  MoveC 574 to (267.87, -55.04, -8.35) mm, rotated rx 180 ry 0 rz 0 deg; joints [19.535, -64.731, 149.655, 19.627, -84.348, -1.431] to (268.06, -55.49, -8.35) mm, rotated rx 180 ry 0 rz 0 deg; joints [19.512, -64.74, 149.678, 19.605, -84.361, -1.424]
  MoveL 575 to (268.06, -80.89, -8.35) mm, rotated rx 180 ry 0 rz 0 deg; joints [18.023, -64.948, 150.269, 18.098, -84.683, -1.18]
  MoveL 576 to (217.26, -80.89, -8.35) mm, rotated rx -180 ry 0 rz 0 deg; joints [17.095, -63.534, 146.744, 17.235, -82.641, -1.736]
  MoveL 577 to (217.26, -30.09, -8.35) mm, rotated rx -180 ry 0 rz 0 deg; joints [19.918, -63.093, 145.562, 20.113, -82.053, -2.311]
  MoveL 578 to (268.06, -30.09, -8.35) mm, rotated rx 180 ry 0 rz 0 deg; joints [20.974, -64.512, 149.041, 21.088, -84.024, -1.694]
  MoveL 579 to (268.06, -55.49, -8.35) mm, rotated rx 180 ry 0 rz 0 deg; joints [19.512, -64.74, 149.678, 19.605, -84.361, -1.424]
  MoveC 580 to (267.87, -55.94, -8.35) mm, rotated rx -180 ry 0 rz 0 deg; joints [19.482, -64.739, 149.677, 19.575, -84.359, -1.422] to (267.42, -56.12, -8.35) mm, rotated rx -180 ry 0 rz 0 deg; joints [19.462, -64.728, 149.65, 19.555, -84.344, -1.425]
  MoveL 581 to (266.79, -56.12, -8.35) mm, rotated rx 180 ry 0 rz 0 deg; joints [19.449, -64.711, 149.607, 19.543, -84.319, -1.433]
  MoveC 582 to (266.34, -56.12, -8.16) mm, rotated rx 180 ry 0 rz 0 deg; joints [19.44, -64.717, 149.577, 19.535, -84.284, -1.445] to (266.15, -56.12, -7.72) mm, rotated rx -180 ry 0 rz 0 deg; joints [19.436, -64.757, 149.566, 19.532, -84.236, -1.461]
  Set speed (500.0 mm/s)
  MoveL 583 to (266.15, -56.12, 6) mm, rotated rx 180 ry 0 rz 0 deg; joints [19.428, -66.123, 149.601, 19.574, -82.982, -1.909]
  MoveL 584 to (139.15, -54.85, 6) mm, rotated rx -180 ry 0 rz 0 deg; joints [17.193, -62.179, 140.681, 17.573, -78.154, -3.178]
  Set speed (25.4 mm/s)
  MoveL 585 to (139.15, -54.85, -3.54) mm, rotated rx 180 ry 0 rz 0 deg; joints [17.198, -61.393, 140.662, 17.531, -78.886, -2.943]
  MoveC 586 to (139.34, -54.85, -3.99) mm, rotated rx 180 ry 0 rz 0 deg; joints [17.201, -61.361, 140.675, 17.531, -78.928, -2.93] to (139.79, -54.85, -4.17) mm, rotated rx 180 ry 0 rz 0 deg; joints [17.208, -61.36, 140.706, 17.537, -78.96, -2.921]
  Set speed (50.8 mm/s)
  MoveL 587 to (140.42, -54.85, -4.17) mm, rotated rx -180 ry 0 rz 0 deg; joints [17.219, -61.38, 140.752, 17.546, -78.985, -2.915]
  MoveC 588 to (140.87, -55.04, -4.17) mm, rotated rx -180 ry 0 rz 0 deg; joints [17.216, -61.395, 140.788, 17.542, -79.004, -2.909] to (141.06, -55.49, -4.17) mm, rotated rx -180 ry 0 rz 0 deg; joints [17.196, -61.405, 140.811, 17.521, -79.016, -2.901]
  MoveL 589 to (141.06, -80.89, -4.17) mm, rotated rx 180 ry 0 rz 0 deg; joints [15.863, -61.621, 141.351, 16.147, -79.257, -2.57]
  MoveL 590 to (90.26, -80.89, -4.17) mm, rotated rx 180 ry 0 rz 0 deg; joints [15.134, -60.003, 137.665, 15.522, -77.228, -3.006]
  MoveL 591 to (90.26, -30.09, -4.17) mm, rotated rx 180 ry 0 rz 0 deg; joints [17.675, -59.554, 136.575, 18.167, -76.776, -3.743]
  MoveL 592 to (141.06, -30.09, -4.18) mm, rotated rx -180 ry 0 rz 0 deg; joints [18.51, -61.17, 140.228, 18.879, -78.762, -3.249]
  MoveL 593 to (141.06, -55.49, -4.17) mm, rotated rx -180 ry 0 rz 0 deg; joints [17.196, -61.405, 140.811, 17.521, -79.016, -2.901]
  MoveC 594 to (140.87, -55.94, -4.17) mm, rotated rx 180 ry 0 rz 0 deg; joints [17.169, -61.403, 140.808, 17.494, -79.013, -2.897] to (140.42, -56.12, -4.18) mm, rotated rx 180 ry 0 rz 0 deg; joints [17.152, -61.391, 140.78, 17.478, -78.997, -2.898]
  MoveL 595 to (139.79, -56.12, -4.18) mm, rotated rx 180 ry 0 rz 0 deg; joints [17.142, -61.371, 140.734, 17.469, -78.972, -2.904]
  MoveC 596 to (139.34, -56.12, -3.99) mm, rotated rx -180 ry 0 rz 0 deg; joints [17.135, -61.373, 140.703, 17.463, -78.94, -2.913] to (139.15, -56.12, -3.54) mm, rotated rx -180 ry 0 rz 0 deg; joints [17.132, -61.404, 140.69, 17.463, -78.899, -2.926]
  Set speed (500.0 mm/s)
  MoveL 597 to (139.15, -56.12, 5) mm, rotated rx -180 ry 0 rz 0 deg; joints [17.128, -62.108, 140.708, 17.5, -78.243, -3.136]
  MoveL 598 to (139.15, -54.85, 5) mm, rotated rx -180 ry 0 rz 0 deg; joints [17.194, -62.097, 140.68, 17.568, -78.231, -3.153]
  Set speed (25.4 mm/s)
  MoveL 599 to (139.15, -54.85, 1.82) mm, rotated rx -180 ry 0 rz 0 deg; joints [17.195, -61.835, 140.674, 17.554, -78.475, -3.075]
  MoveL 600 to (139.15, -54.85, -7.71) mm, rotated rx -180 ry 0 rz 0 deg; joints [17.2, -61.047, 140.651, 17.513, -79.205, -2.841]
  MoveC 601 to (139.34, -54.85, -8.16) mm, rotated rx -180 ry 0 rz 0 deg; joints [17.203, -61.016, 140.663, 17.514, -79.247, -2.828] to (139.79, -54.85, -8.35) mm, rotated rx -180 ry 0 rz 0 deg; joints [17.21, -61.014, 140.695, 17.52, -79.279, -2.819]
  Set speed (50.8 mm/s)
  MoveL 602 to (140.42, -54.85, -8.35) mm, rotated rx -180 ry 0 rz 0 deg; joints [17.221, -61.034, 140.74, 17.529, -79.304, -2.813]
  MoveC 603 to (140.87, -55.04, -8.35) mm, rotated rx 180 ry 0 rz 0 deg; joints [17.218, -61.049, 140.776, 17.525, -79.324, -2.806] to (141.06, -55.49, -8.35) mm, rotated rx 180 ry 0 rz 0 deg; joints [17.198, -61.059, 140.8, 17.503, -79.336, -2.799]
  MoveL 604 to (141.06, -80.89, -8.35) mm, rotated rx -180 ry 0 rz 0 deg; joints [15.865, -61.271, 141.339, 16.132, -79.582, -2.475]
  MoveL 605 to (90.26, -80.89, -8.35) mm, rotated rx -180 ry 0 rz 0 deg; joints [15.136, -59.676, 137.654, 15.505, -77.533, -2.92]
  MoveL 606 to (90.26, -30.09, -8.35) mm, rotated rx -180 ry 0 rz 0 deg; joints [17.677, -59.233, 136.564, 18.146, -77.071, -3.645]
  MoveL 607 to (141.06, -30.09, -8.35) mm, rotated rx 180 ry 0 rz 0 deg; joints [18.512, -60.828, 140.217, 18.86, -79.076, -3.141]
  MoveL 608 to (141.06, -55.49, -8.35) mm, rotated rx 180 ry 0 rz 0 deg; joints [17.198, -61.059, 140.8, 17.503, -79.336, -2.799]
  MoveC 609 to (140.87, -55.94, -8.35) mm, rotated rx -180 ry 0 rz 0 deg; joints [17.171, -61.057, 140.796, 17.477, -79.333, -2.795] to (140.42, -56.12, -8.35) mm, rotated rx 180 ry 0 rz 0 deg; joints [17.155, -61.045, 140.768, 17.46, -79.317, -2.796]
  MoveL 610 to (139.79, -56.12, -8.35) mm, rotated rx 180 ry 0 rz 0 deg; joints [17.144, -61.025, 140.723, 17.452, -79.291, -2.803]
  MoveC 611 to (139.34, -56.12, -8.16) mm, rotated rx -180 ry 0 rz 0 deg; joints [17.137, -61.027, 140.691, 17.446, -79.259, -2.811] to (139.15, -56.12, -7.72) mm, rotated rx -180 ry 0 rz 0 deg; joints [17.134, -61.058, 140.679, 17.445, -79.218, -2.824]
  Set speed (500.0 mm/s)
  MoveL 612 to (139.15, -56.12, 6) mm, rotated rx -180 ry 0 rz 0 deg; joints [17.127, -62.191, 140.709, 17.505, -78.166, -3.16]
  MoveL 613 to (139.15, -235.88, 6) mm, rotated rx -180 ry 0 rz 0 deg; joints [7.369, -63.345, 143.558, 7.492, -79.426, -0.998]
  Set speed (25.4 mm/s)
  MoveL 614 to (139.15, -235.88, -3.54) mm, rotated rx 180 ry 0 rz 0 deg; joints [7.373, -62.513, 143.538, 7.477, -80.231, -0.891]
  MoveC 615 to (139.34, -235.88, -3.99) mm, rotated rx -180 ry 0 rz 0 deg; joints [7.374, -62.48, 143.551, 7.477, -80.276, -0.885] to (139.79, -235.88, -4.17) mm, rotated rx -180 ry 0 rz 0 deg; joints [7.378, -62.477, 143.583, 7.48, -80.311, -0.881]
  Set speed (50.8 mm/s)
  MoveL 616 to (140.42, -235.88, -4.18) mm, rotated rx -180 ry 0 rz 0 deg; joints [7.382, -62.497, 143.63, 7.484, -80.337, -0.878]
  MoveC 617 to (140.87, -236.07, -4.18) mm, rotated rx -180 ry 0 rz 0 deg; joints [7.375, -62.512, 143.665, 7.476, -80.357, -0.874] to (141.06, -236.52, -4.18) mm, rotated rx -180 ry 0 rz 0 deg; joints [7.351, -62.519, 143.683, 7.452, -80.367, -0.869]
  MoveL 618 to (141.06, -261.92, -4.17) mm, rotated rx 180 ry 0 rz 0 deg; joints [5.92, -62.597, 143.899, 5.998, -80.48, -0.633]
  MoveL 619 to (90.26, -261.92, -4.18) mm, rotated rx -180 ry 0 rz 0 deg; joints [5.637, -60.978, 140.132, 5.751, -78.337, -0.808]
  MoveL 620 to (90.26, -211.12, -4.17) mm, rotated rx 180 ry 0 rz 0 deg; joints [8.357, -60.803, 139.668, 8.536, -78.115, -1.37]
  MoveL 621 to (141.06, -211.12, -4.17) mm, rotated rx -180 ry 0 rz 0 deg; joints [8.773, -62.422, 143.419, 8.898, -80.234, -1.115]
  MoveL 622 to (141.06, -236.52, -4.18) mm, rotated rx -180 ry 0 rz 0 deg; joints [7.351, -62.519, 143.683, 7.452, -80.367, -0.869]
  MoveC 623 to (140.87, -236.97, -4.17) mm, rotated rx -180 ry 0 rz 0 deg; joints [7.325, -62.515, 143.673, 7.425, -80.362, -0.866] to (140.42, -237.16, -4.17) mm, rotated rx -180 ry 0 rz 0 deg; joints [7.311, -62.502, 143.642, 7.412, -80.344, -0.866]
  MoveL 624 to (139.79, -237.16, -4.17) mm, rotated rx 180 ry 0 rz 0 deg; joints [7.306, -62.482, 143.595, 7.408, -80.317, -0.869]
  MoveC 625 to (139.34, -237.15, -3.99) mm, rotated rx -180 ry 0 rz 0 deg; joints [7.303, -62.484, 143.563, 7.405, -80.282, -0.873] to (139.15, -237.15, -3.54) mm, rotated rx -180 ry 0 rz 0 deg; joints [7.302, -62.517, 143.55, 7.404, -80.237, -0.879]
  Set speed (500.0 mm/s)
  MoveL 626 to (139.15, -237.16, 5) mm, rotated rx 180 ry 0 rz 0 deg; joints [7.298, -63.263, 143.569, 7.418, -79.516, -0.973]
  MoveL 627 to (139.15, -235.88, 5) mm, rotated rx -180 ry 0 rz 0 deg; joints [7.37, -63.258, 143.557, 7.491, -79.51, -0.987]
  Set speed (25.4 mm/s)
  MoveL 628 to (139.15, -235.89, 1.82) mm, rotated rx 180 ry 0 rz 0 deg; joints [7.371, -62.981, 143.551, 7.485, -79.779, -0.951]
  MoveL 629 to (139.15, -235.88, -7.71) mm, rotated rx -180 ry 0 rz 0 deg; joints [7.374, -62.148, 143.526, 7.471, -80.581, -0.845]
  MoveC 630 to (139.34, -235.88, -8.16) mm, rotated rx -180 ry 0 rz 0 deg; joints [7.376, -62.114, 143.539, 7.471, -80.627, -0.839] to (139.79, -235.89, -8.35) mm, rotated rx 180 ry 0 rz 0 deg; joints [7.379, -62.111, 143.571, 7.474, -80.661, -0.835]
  Set speed (50.8 mm/s)
  MoveL 631 to (140.42, -235.88, -8.35) mm, rotated rx -180 ry 0 rz 0 deg; joints [7.384, -62.131, 143.618, 7.478, -80.688, -0.832]
  MoveC 632 to (140.87, -236.07, -8.35) mm, rotated rx -180 ry 0 rz 0 deg; joints [7.377, -62.145, 143.652, 7.47, -80.708, -0.828] to (141.06, -236.52, -8.35) mm, rotated rx -180 ry 0 rz 0 deg; joints [7.353, -62.153, 143.67, 7.446, -80.718, -0.823]
  MoveL 633 to (141.06, -261.92, -8.35) mm, rotated rx -180 ry 0 rz 0 deg; joints [5.921, -62.229, 143.887, 5.993, -80.834, -0.596]
  MoveL 634 to (90.26, -261.92, -8.35) mm, rotated rx -180 ry 0 rz 0 deg; joints [5.638, -60.636, 140.12, 5.746, -78.666, -0.775]
  MoveL 635 to (90.26, -211.12, -8.35) mm, rotated rx 180 ry 0 rz 0 deg; joints [8.358, -60.464, 139.657, 8.528, -78.439, -1.321]
  MoveL 636 to (141.06, -211.12, -8.35) mm, rotated rx 180 ry 0 rz 0 deg; joints [8.775, -62.058, 143.407, 8.891, -80.582, -1.06]
  MoveL 637 to (141.06, -236.52, -8.35) mm, rotated rx -180 ry 0 rz 0 deg; joints [7.353, -62.153, 143.67, 7.446, -80.718, -0.823]
  MoveC 638 to (140.87, -236.97, -8.35) mm, rotated rx 180 ry 0 rz 0 deg; joints [7.326, -62.148, 143.661, 7.419, -80.713, -0.82] to (140.42, -237.16, -8.35) mm, rotated rx -180 ry 0 rz 0 deg; joints [7.313, -62.135, 143.63, 7.406, -80.695, -0.82]
  MoveL 639 to (139.79, -237.15, -8.35) mm, rotated rx -180 ry 0 rz 0 deg; joints [7.308, -62.116, 143.583, 7.402, -80.668, -0.823]
  MoveC 640 to (139.34, -237.15, -8.16) mm, rotated rx 180 ry 0 rz 0 deg; joints [7.305, -62.118, 143.551, 7.399, -80.633, -0.827] to (139.15, -237.16, -7.72) mm, rotated rx -180 ry 0 rz 0 deg; joints [7.303, -62.152, 143.538, 7.398, -80.587, -0.833]
  Set speed (500.0 mm/s)
  MoveL 641 to (139.15, -237.16, 6) mm, rotated rx -180 ry 0 rz 0 deg; joints [7.298, -63.35, 143.57, 7.42, -79.431, -0.985]
  MoveL 642 to (266.15, -235.88, 6) mm, rotated rx -180 ry 0 rz 0 deg; joints [8.42, -67.287, 152.736, 8.452, -84.629, -0.396]
  Set speed (25.4 mm/s)
  MoveL 643 to (266.15, -235.89, -3.54) mm, rotated rx 180 ry 0 rz 0 deg; joints [8.424, -66.261, 152.712, 8.444, -85.619, -0.249]
  MoveC 644 to (266.34, -235.88, -3.99) mm, rotated rx -180 ry 0 rz 0 deg; joints [8.426, -66.218, 152.723, 8.445, -85.674, -0.241] to (266.79, -235.89, -4.17) mm, rotated rx -180 ry 0 rz 0 deg; joints [8.43, -66.21, 152.755, 8.449, -85.712, -0.235]
  Set speed (50.8 mm/s)
  MoveL 645 to (267.42, -235.89, -4.17) mm, rotated rx -180 ry 0 rz 0 deg; joints [8.436, -66.228, 152.8, 8.455, -85.74, -0.231]
  MoveC 646 to (267.87, -236.07, -4.18) mm, rotated rx -180 ry 0 rz 0 deg; joints [8.429, -66.241, 152.834, 8.447, -85.76, -0.228] to (268.06, -236.52, -4.17) mm, rotated rx 180 ry 0 rz 0 deg; joints [8.402, -66.247, 152.852, 8.42, -85.772, -0.225]
  MoveL 647 to (268.06, -261.92, -4.18) mm, rotated rx -180 ry 0 rz 0 deg; joints [6.77, -66.321, 153.092, 6.782, -85.924, -0.109]
  MoveL 648 to (217.26, -261.92, -4.18) mm, rotated rx 180 ry 0 rz 0 deg; joints [6.402, -64.892, 149.45, 6.436, -83.722, -0.337]
  MoveL 649 to (217.26, -211.12, -4.18) mm, rotated rx -180 ry 0 rz 0 deg; joints [9.482, -64.721, 148.941, 9.54, -83.43, -0.684]
  MoveL 650 to (268.06, -211.12, -4.17) mm, rotated rx 180 ry 0 rz 0 deg; joints [10.02, -66.154, 152.56, 10.045, -85.591, -0.354]
  MoveL 651 to (268.06, -236.52, -4.17) mm, rotated rx 180 ry 0 rz 0 deg; joints [8.402, -66.247, 152.852, 8.42, -85.772, -0.225]
  MoveC 652 to (267.87, -236.97, -4.17) mm, rotated rx -180 ry 0 rz 0 deg; joints [8.371, -66.244, 152.843, 8.389, -85.766, -0.224] to (267.42, -237.15, -4.18) mm, rotated rx -180 ry 0 rz 0 deg; joints [8.355, -66.232, 152.813, 8.373, -85.748, -0.225]
  MoveL 653 to (266.79, -237.15, -4.18) mm, rotated rx -180 ry 0 rz 0 deg; joints [8.349, -66.215, 152.768, 8.368, -85.721, -0.229]
  MoveC 654 to (266.34, -237.15, -3.99) mm, rotated rx 180 ry 0 rz 0 deg; joints [8.345, -66.222, 152.737, 8.364, -85.682, -0.234] to (266.15, -237.16, -3.54) mm, rotated rx 180 ry 0 rz 0 deg; joints [8.343, -66.266, 152.725, 8.362, -85.627, -0.242]
  Set speed (500.0 mm/s)
  MoveL 655 to (266.15, -237.16, 5) mm, rotated rx -180 ry 0 rz 0 deg; joints [8.339, -67.184, 152.747, 8.37, -84.741, -0.373]
  MoveL 656 to (266.15, -235.89, 5) mm, rotated rx -180 ry 0 rz 0 deg; joints [8.42, -67.18, 152.734, 8.451, -84.733, -0.38]
  Set speed (25.4 mm/s)
  MoveL 657 to (266.15, -235.88, 1.82) mm, rotated rx -180 ry 0 rz 0 deg; joints [8.422, -66.839, 152.727, 8.448, -85.063, -0.331]
  MoveL 658 to (266.15, -235.89, -7.71) mm, rotated rx 180 ry 0 rz 0 deg; joints [8.426, -65.811, 152.697, 8.441, -86.05, -0.185]
  MoveC 659 to (266.34, -235.89, -8.16) mm, rotated rx -180 ry 0 rz 0 deg; joints [8.428, -65.768, 152.709, 8.442, -86.104, -0.177] to (266.79, -235.88, -8.35) mm, rotated rx -180 ry 0 rz 0 deg; joints [8.432, -65.76, 152.74, 8.446, -86.143, -0.171]
  Set speed (50.8 mm/s)
  MoveL 660 to (267.42, -235.88, -8.35) mm, rotated rx -180 ry 0 rz 0 deg; joints [8.438, -65.777, 152.785, 8.452, -86.171, -0.167]
  MoveC 661 to (267.87, -236.07, -8.35) mm, rotated rx 180 ry 0 rz 0 deg; joints [8.431, -65.789, 152.819, 8.444, -86.193, -0.164] to (268.06, -236.52, -8.35) mm, rotated rx 180 ry 0 rz 0 deg; joints [8.404, -65.795, 152.837, 8.417, -86.204, -0.161]
  MoveL 662 to (268.06, -261.92, -8.35) mm, rotated rx -180 ry 0 rz 0 deg; joints [6.772, -65.866, 153.077, 6.781, -86.361, -0.057]
  MoveL 663 to (217.26, -261.92, -8.35) mm, rotated rx 180 ry 0 rz 0 deg; joints [6.404, -64.477, 149.436, 6.433, -84.122, -0.292]
  MoveL 664 to (217.26, -211.12, -8.35) mm, rotated rx 180 ry 0 rz 0 deg; joints [9.483, -64.31, 148.928, 9.534, -83.822, -0.618]
  MoveL 665 to (268.06, -211.12, -8.35) mm, rotated rx -180 ry 0 rz 0 deg; joints [10.022, -65.706, 152.546, 10.041, -86.018, -0.278]
  MoveL 666 to (268.06, -236.52, -8.35) mm, rotated rx -180 ry 0 rz 0 deg; joints [8.404, -65.795, 152.837, 8.417, -86.204, -0.161]
  MoveC 667 to (267.87, -236.97, -8.35) mm, rotated rx -180 ry 0 rz 0 deg; joints [8.373, -65.792, 152.828, 8.387, -86.199, -0.16] to (267.42, -237.15, -8.35) mm, rotated rx -180 ry 0 rz 0 deg; joints [8.357, -65.781, 152.798, 8.371, -86.18, -0.162]
  MoveL 668 to (266.79, -237.15, -8.35) mm, rotated rx -180 ry 0 rz 0 deg; joints [8.351, -65.764, 152.753, 8.365, -86.152, -0.165]
  MoveC 669 to (266.34, -237.15, -8.16) mm, rotated rx -180 ry 0 rz 0 deg; joints [8.347, -65.772, 152.722, 8.361, -86.113, -0.171] to (266.15, -237.15, -7.72) mm, rotated rx 180 ry 0 rz 0 deg; joints [8.345, -65.815, 152.711, 8.36, -86.059, -0.179]
  Set speed (500.0 mm/s)
  MoveL 670 to (266.15, -237.15, 6) mm, rotated rx -180 ry 0 rz 0 deg; joints [8.339, -67.291, 152.749, 8.371, -84.636, -0.388]
  MoveL 671 to (393.15, -235.89, 6) mm, rotated rx 180 ry 0 rz 30 deg; joints [20.408, -68.62, 155.616, 50.482, -87.198, -2.516]
  Set speed (25.4 mm/s)
  MoveL 672 to (393.15, -235.88, -3.54) mm, rotated rx -180 ry 0 rz 30 deg; joints [20.414, -67.513, 155.591, 50.452, -87.887, -1.681]
  MoveC 673 to (393.34, -235.89, -3.99) mm, rotated rx 180 ry 0 rz 30 deg; joints [20.419, -67.465, 155.602, 50.455, -87.924, -1.636] to (393.79, -235.88, -4.17) mm, rotated rx -180 ry 0 rz 30 deg; joints [20.43, -67.455, 155.631, 50.465, -87.95, -1.605]
  Set speed (50.8 mm/s)
  MoveL 674 to (394.42, -235.88, -4.18) mm, rotated rx -180 ry 0 rz 30 deg; joints [20.445, -67.47, 155.674, 50.479, -87.967, -1.585]
  MoveC 675 to (394.87, -236.07, -4.17) mm, rotated rx -180 ry 0 rz 30 deg; joints [20.443, -67.483, 155.708, 50.478, -87.981, -1.568] to (395.06, -236.52, -4.18) mm, rotated rx -180 ry 0 rz 30 deg; joints [20.419, -67.491, 155.732, 50.453, -87.99, -1.555]
  MoveL 676 to (395.06, -261.92, -4.17) mm, rotated rx -180 ry 0 rz 30 deg; joints [18.79, -67.683, 156.338, 48.813, -88.225, -1.211]
  MoveL 677 to (344.26, -261.92, -4.18) mm, rotated rx -180 ry 0 rz 30 deg; joints [17.731, -66.386, 152.89, 47.824, -86.761, -2.789]
  MoveL 678 to (344.26, -211.12, -4.17) mm, rotated rx 180 ry 0 rz 0 deg; joints [10.952, -68.118, 157.906, 10.948, -88.922, 0.232]
  MoveL 679 to (395.06, -211.12, -4.18) mm, rotated rx -180 ry 0 rz 30 deg; joints [22.015, -67.278, 155.078, 52.062, -87.757, -1.935]
  MoveL 680 to (395.06, -236.52, -4.17) mm, rotated rx -180 ry 0 rz 30 deg; joints [20.419, -67.491, 155.732, 50.453, -87.99, -1.555]
  MoveC 681 to (394.87, -236.97, -4.18) mm, rotated rx 180 ry 0 rz 30 deg; joints [20.386, -67.49, 155.731, 50.42, -87.989, -1.555] to (394.42, -237.15, -4.18) mm, rotated rx -180 ry 0 rz 30 deg; joints [20.364, -67.48, 155.705, 50.398, -87.979, -1.567]
  MoveL 682 to (393.79, -237.16, -4.18) mm, rotated rx 180 ry 0 rz 30 deg; joints [20.349, -67.465, 155.663, 50.384, -87.961, -1.587]
  MoveC 683 to (393.34, -237.15, -3.99) mm, rotated rx -180 ry 0 rz 30 deg; joints [20.338, -67.475, 155.634, 50.374, -87.936, -1.618] to (393.15, -237.15, -3.54) mm, rotated rx 180 ry 0 rz 30 deg; joints [20.334, -67.523, 155.623, 50.371, -87.898, -1.663]
  Set speed (500.0 mm/s)
  MoveL 684 to (393.15, -237.16, 5) mm, rotated rx -180 ry 0 rz 30 deg; joints [20.328, -68.515, 155.646, 50.397, -87.28, -2.41]
  MoveL 685 to (393.15, -235.88, 5) mm, rotated rx 180 ry 0 rz 30 deg; joints [20.408, -68.504, 155.614, 50.478, -87.27, -2.428]
  Set speed (25.4 mm/s)
  MoveL 686 to (393.15, -235.88, 1.82) mm, rotated rx -180 ry 0 rz 30 deg; joints [20.411, -68.136, 155.607, 50.468, -87.5, -2.15]
  MoveL 687 to (393.15, -235.89, -7.71) mm, rotated rx -180 ry 0 rz 30 deg; joints [20.417, -67.027, 155.576, 50.443, -88.187, -1.318]
  MoveC 688 to (393.34, -235.89, -8.16) mm, rotated rx 180 ry 0 rz 30 deg; joints [20.422, -66.979, 155.587, 50.446, -88.224, -1.272] to (393.79, -235.88, -8.35) mm, rotated rx -180 ry 0 rz 30 deg; joints [20.432, -66.968, 155.616, 50.456, -88.25, -1.242]
  Set speed (50.8 mm/s)
  MoveL 689 to (394.42, -235.89, -8.35) mm, rotated rx 180 ry 0 rz 30 deg; joints [20.447, -66.983, 155.658, 50.47, -88.267, -1.221]
  MoveC 690 to (394.87, -236.07, -8.35) mm, rotated rx -180 ry 0 rz 30 deg; joints [20.446, -66.995, 155.693, 50.468, -88.282, -1.203] to (395.06, -236.52, -8.35) mm, rotated rx -180 ry 0 rz 30 deg; joints [20.422, -67.003, 155.717, 50.444, -88.291, -1.191]
  MoveL 691 to (395.06, -261.92, -8.35) mm, rotated rx -180 ry 0 rz 30 deg; joints [18.792, -67.187, 156.322, 48.805, -88.541, -0.85]
  MoveL 692 to (344.26, -261.92, -8.35) mm, rotated rx -180 ry 0 rz 30 deg; joints [17.733, -65.934, 152.875, 47.809, -87.055, -2.465]
  MoveL 693 to (344.26, -211.12, -8.35) mm, rotated rx -180 ry 0 rz 0 deg; joints [10.954, -67.598, 157.889, 10.949, -89.416, 0.328]
  MoveL 694 to (395.06, -211.12, -8.35) mm, rotated rx -180 ry 0 rz 30 deg; joints [22.018, -66.799, 155.062, 52.051, -88.042, -1.568]
  MoveL 695 to (395.06, -236.52, -8.35) mm, rotated rx -180 ry 0 rz 30 deg; joints [20.422, -67.003, 155.717, 50.444, -88.291, -1.191]
  MoveC 696 to (394.87, -236.97, -8.35) mm, rotated rx -180 ry 0 rz 30 deg; joints [20.389, -67.002, 155.715, 50.411, -88.291, -1.191] to (394.42, -237.15, -8.35) mm, rotated rx 180 ry 0 rz 30 deg; joints [20.367, -66.993, 155.69, 50.389, -88.28, -1.203]
  MoveL 697 to (393.79, -237.15, -8.35) mm, rotated rx -180 ry 0 rz 30 deg; joints [20.352, -66.978, 155.648, 50.375, -88.262, -1.224]
  MoveC 698 to (393.34, -237.15, -8.16) mm, rotated rx -180 ry 0 rz 30 deg; joints [20.341, -66.989, 155.618, 50.365, -88.236, -1.254] to (393.15, -237.15, -7.72) mm, rotated rx 180 ry 0 rz 30 deg; joints [20.336, -67.037, 155.608, 50.362, -88.199, -1.3]
  Set speed (500.0 mm/s)
  MoveL 699 to (393.15, -237.16, 6) mm, rotated rx -180 ry 0 rz 30 deg; joints [20.327, -68.631, 155.648, 50.401, -87.207, -2.498]
  MoveL 700 to (393.15, -422.22, 6) mm, rotated rx -180 ry 0 rz 60 deg; joints [14.177, -65.672, 148.72, 74.367, -87.443, -7.311]
  Set speed (25.4 mm/s)
  MoveL 701 to (393.15, -422.22, -3.54) mm, rotated rx -180 ry 0 rz 60 deg; joints [14.182, -64.742, 148.698, 74.335, -87.688, -6.436]
  MoveC 702 to (393.34, -422.22, -3.99) mm, rotated rx -180 ry 0 rz 60 deg; joints [14.185, -64.704, 148.71, 74.336, -87.702, -6.387] to (393.79, -422.22, -4.17) mm, rotated rx -180 ry 0 rz 60 deg; joints [14.192, -64.698, 148.741, 74.342, -87.713, -6.353]
  Set speed (50.8 mm/s)
  MoveL 703 to (394.42, -422.22, -4.18) mm, rotated rx -180 ry 0 rz 60 deg; joints [14.201, -64.717, 148.786, 74.35, -87.721, -6.327]
  MoveC 704 to (394.87, -422.41, -4.18) mm, rotated rx -180 ry 0 rz 60 deg; joints [14.197, -64.731, 148.821, 74.345, -87.726, -6.307] to (395.06, -422.86, -4.17) mm, rotated rx -180 ry 0 rz 60 deg; joints [14.173, -64.739, 148.842, 74.321, -87.727, -6.294]
  MoveL 705 to (395.06, -448.26, -4.17) mm, rotated rx -180 ry 0 rz 60 deg; joints [12.665, -64.892, 149.27, 72.807, -87.66, -5.987]
  MoveL 706 to (344.26, -448.26, -4.17) mm, rotated rx -180 ry 0 rz 30 deg; joints [5.639, -67.24, 155.598, 35.664, -87.777, -1.156]
  MoveL 707 to (344.26, -397.46, -4.18) mm, rotated rx 180 ry 0 rz 30 deg; joints [9.034, -67.111, 155.137, 39.069, -87.578, -1.443]
  MoveL 708 to (395.06, -397.46, -4.17) mm, rotated rx 180 ry 0 rz 60 deg; joints [15.662, -64.566, 148.367, 75.814, -87.801, -6.627]
  MoveL 709 to (395.06, -422.86, -4.17) mm, rotated rx -180 ry 0 rz 60 deg; joints [14.173, -64.739, 148.842, 74.321, -87.727, -6.294]
  MoveC 710 to (394.87, -423.31, -4.18) mm, rotated rx -180 ry 0 rz 60 deg; joints [14.144, -64.737, 148.837, 74.292, -87.724, -6.296] to (394.42, -423.49, -4.18) mm, rotated rx 180 ry 0 rz 60 deg; joints [14.126, -64.725, 148.809, 74.275, -87.717, -6.311]
  MoveL 711 to (393.79, -423.49, -4.17) mm, rotated rx -180 ry 0 rz 60 deg; joints [14.117, -64.707, 148.764, 74.266, -87.709, -6.337]
  MoveC 712 to (393.34, -423.49, -3.99) mm, rotated rx -180 ry 0 rz 60 deg; joints [14.11, -64.712, 148.733, 74.261, -87.699, -6.372] to (393.15, -423.49, -3.54) mm, rotated rx -180 ry 0 rz 60 deg; joints [14.107, -64.75, 148.721, 74.26, -87.685, -6.42]
  Set speed (500.0 mm/s)
  MoveL 713 to (393.15, -423.49, 5) mm, rotated rx -180 ry 0 rz 60 deg; joints [14.103, -65.583, 148.741, 74.289, -87.464, -7.203]
  MoveL 714 to (393.15, -422.22, 5) mm, rotated rx 180 ry 0 rz 60 deg; joints [14.178, -65.575, 148.718, 74.364, -87.469, -7.219]
  Set speed (25.4 mm/s)
  MoveL 715 to (393.15, -422.22, 1.82) mm, rotated rx 180 ry 0 rz 60 deg; joints [14.179, -65.266, 148.712, 74.353, -87.551, -6.927]
  MoveL 716 to (393.15, -422.22, -7.71) mm, rotated rx -180 ry 0 rz 60 deg; joints [14.184, -64.334, 148.685, 74.322, -87.795, -6.055]
  MoveC 717 to (393.34, -422.22, -8.16) mm, rotated rx 180 ry 0 rz 60 deg; joints [14.187, -64.295, 148.697, 74.323, -87.809, -6.007] to (393.79, -422.22, -8.35) mm, rotated rx 180 ry 0 rz 60 deg; joints [14.194, -64.29, 148.728, 74.329, -87.82, -5.972]
  Set speed (50.8 mm/s)
  MoveL 718 to (394.42, -422.22, -8.35) mm, rotated rx -180 ry 0 rz 60 deg; joints [14.203, -64.308, 148.773, 74.337, -87.828, -5.946]
  MoveC 719 to (394.87, -422.41, -8.35) mm, rotated rx -180 ry 0 rz 60 deg; joints [14.199, -64.321, 148.808, 74.332, -87.833, -5.925] to (395.06, -422.86, -8.35) mm, rotated rx -180 ry 0 rz 60 deg; joints [14.175, -64.329, 148.829, 74.308, -87.835, -5.912]
  MoveL 720 to (395.06, -448.26, -8.35) mm, rotated rx -180 ry 0 rz 60 deg; joints [12.667, -64.478, 149.256, 72.794, -87.778, -5.605]
  MoveL 721 to (344.26, -448.26, -8.35) mm, rotated rx -180 ry 0 rz 30 deg; joints [5.641, -66.754, 155.583, 35.656, -88.159, -0.882]
  MoveL 722 to (344.26, -397.46, -8.35) mm, rotated rx -180 ry 0 rz 30 deg; joints [9.036, -66.631, 155.122, 39.06, -87.939, -1.15]
  MoveL 723 to (395.06, -397.46, -8.35) mm, rotated rx -180 ry 0 rz 60 deg; joints [15.664, -64.161, 148.354, 75.802, -87.897, -6.247]
  MoveL 724 to (395.06, -422.86, -8.35) mm, rotated rx -180 ry 0 rz 60 deg; joints [14.175, -64.329, 148.829, 74.308, -87.835, -5.912]
  MoveC 725 to (394.87, -423.31, -8.35) mm, rotated rx -180 ry 0 rz 60 deg; joints [14.146, -64.327, 148.824, 74.279, -87.831, -5.914] to (394.42, -423.49, -8.35) mm, rotated rx -180 ry 0 rz 60 deg; joints [14.128, -64.315, 148.795, 74.262, -87.825, -5.93]
  MoveL 726 to (393.79, -423.49, -8.35) mm, rotated rx -180 ry 0 rz 60 deg; joints [14.119, -64.298, 148.75, 74.254, -87.817, -5.956]
  MoveC 727 to (393.34, -423.49, -8.16) mm, rotated rx -180 ry 0 rz 60 deg; joints [14.112, -64.303, 148.719, 74.248, -87.806, -5.991] to (393.15, -423.49, -7.72) mm, rotated rx -180 ry 0 rz 60 deg; joints [14.109, -64.342, 148.708, 74.247, -87.792, -6.039]
  Set speed (500.0 mm/s)
  MoveL 728 to (393.15, -423.49, 6) mm, rotated rx -180 ry 0 rz 60 deg; joints [14.102, -65.681, 148.743, 74.293, -87.438, -7.295]
  MoveL 729 to (266.15, -422.22, 6) mm, rotated rx -180 ry 0 rz 0 deg; joints [-3.67, -67.406, 153.291, -3.688, -85.023, 0.537]
  Set speed (25.4 mm/s)
  MoveL 730 to (266.15, -422.22, -3.54) mm, rotated rx 180 ry 0 rz 0 deg; joints [-3.668, -66.366, 153.266, -3.681, -86.037, 0.471]
  MoveC 731 to (266.34, -422.22, -3.99) mm, rotated rx -180 ry 0 rz 0 deg; joints [-3.669, -66.322, 153.277, -3.681, -86.092, 0.468] to (266.79, -422.22, -4.17) mm, rotated rx 180 ry 0 rz 0 deg; joints [-3.671, -66.314, 153.309, -3.683, -86.132, 0.465]
  Set speed (50.8 mm/s)
  MoveL 732 to (267.42, -422.22, -4.18) mm, rotated rx 180 ry 0 rz 0 deg; joints [-3.673, -66.331, 153.354, -3.685, -86.16, 0.464]
  MoveC 733 to (267.87, -422.41, -4.18) mm, rotated rx -180 ry 0 rz 0 deg; joints [-3.687, -66.343, 153.386, -3.699, -86.18, 0.463] to (268.06, -422.86, -4.18) mm, rotated rx 180 ry 0 rz 0 deg; joints [-3.717, -66.347, 153.397, -3.729, -86.187, 0.464]
  MoveL 734 to (268.06, -448.26, -4.17) mm, rotated rx 180 ry 0 rz 0 deg; joints [-5.368, -66.282, 153.252, -5.384, -86.114, 0.557]
  MoveL 735 to (217.26, -448.26, -4.17) mm, rotated rx -180 ry 0 rz 0 deg; joints [-5.075, -64.863, 149.604, -5.108, -83.891, 0.74]
  MoveL 736 to (217.26, -397.46, -4.18) mm, rotated rx -180 ry 0 rz 0 deg; joints [-1.948, -64.973, 149.83, -1.962, -83.991, 0.448]
  MoveL 737 to (268.06, -397.46, -4.17) mm, rotated rx -180 ry 0 rz 0 deg; joints [-2.061, -66.392, 153.489, -2.069, -86.229, 0.377]
  MoveL 738 to (268.06, -422.86, -4.18) mm, rotated rx 180 ry 0 rz 0 deg; joints [-3.717, -66.347, 153.397, -3.729, -86.187, 0.464]
  MoveC 739 to (267.87, -423.31, -4.18) mm, rotated rx 180 ry 0 rz 0 deg; joints [-3.746, -66.341, 153.382, -3.758, -86.178, 0.466] to (267.42, -423.49, -4.18) mm, rotated rx -180 ry 0 rz 0 deg; joints [-3.756, -66.328, 153.348, -3.768, -86.157, 0.468]
  MoveL 740 to (266.79, -423.49, -4.18) mm, rotated rx -180 ry 0 rz 0 deg; joints [-3.753, -66.311, 153.303, -3.766, -86.129, 0.47]
  MoveC 741 to (266.34, -423.49, -3.99) mm, rotated rx -180 ry 0 rz 0 deg; joints [-3.751, -66.319, 153.272, -3.764, -86.089, 0.472] to (266.15, -423.49, -3.54) mm, rotated rx -180 ry 0 rz 0 deg; joints [-3.751, -66.363, 153.26, -3.763, -86.034, 0.476]
  Set speed (500.0 mm/s)
  MoveL 742 to (266.15, -423.49, 5) mm, rotated rx -180 ry 0 rz 0 deg; joints [-3.753, -67.295, 153.283, -3.77, -85.127, 0.536]
  MoveL 743 to (266.15, -422.22, 5) mm, rotated rx -180 ry 0 rz 0 deg; joints [-3.67, -67.298, 153.288, -3.687, -85.13, 0.53]
  Set speed (25.4 mm/s)
  MoveL 744 to (266.15, -422.22, 1.82) mm, rotated rx -180 ry 0 rz 0 deg; joints [-3.669, -66.952, 153.281, -3.685, -85.468, 0.508]
  MoveL 745 to (266.15, -422.22, -7.71) mm, rotated rx -180 ry 0 rz 0 deg; joints [-3.667, -65.909, 153.251, -3.678, -86.477, 0.443]
  MoveC 746 to (266.34, -422.22, -8.16) mm, rotated rx 180 ry 0 rz 0 deg; joints [-3.668, -65.865, 153.262, -3.678, -86.533, 0.439] to (266.79, -422.22, -8.35) mm, rotated rx -180 ry 0 rz 0 deg; joints [-3.67, -65.857, 153.294, -3.68, -86.573, 0.437]
  Set speed (50.8 mm/s)
  MoveL 747 to (267.42, -422.22, -8.35) mm, rotated rx 180 ry 0 rz 0 deg; joints [-3.672, -65.873, 153.339, -3.682, -86.602, 0.435]
  MoveC 748 to (267.87, -422.41, -8.35) mm, rotated rx 180 ry 0 rz 0 deg; joints [-3.686, -65.884, 153.371, -3.696, -86.622, 0.434] to (268.06, -422.86, -8.35) mm, rotated rx -180 ry 0 rz 0 deg; joints [-3.716, -65.888, 153.382, -3.726, -86.629, 0.435]
  MoveL 749 to (268.06, -448.26, -8.35) mm, rotated rx 180 ry 0 rz 0 deg; joints [-5.367, -65.826, 153.237, -5.38, -86.553, 0.515]
  MoveL 750 to (217.26, -448.26, -8.35) mm, rotated rx -180 ry 0 rz 0 deg; joints [-5.074, -64.446, 149.59, -5.103, -84.293, 0.704]
  MoveL 751 to (217.26, -397.46, -8.35) mm, rotated rx -180 ry 0 rz 0 deg; joints [-1.947, -64.553, 149.816, -1.96, -84.396, 0.434]
  MoveL 752 to (268.06, -397.46, -8.35) mm, rotated rx 180 ry 0 rz 0 deg; joints [-2.06, -65.933, 153.474, -2.067, -86.673, 0.361]
  MoveL 753 to (268.06, -422.86, -8.35) mm, rotated rx -180 ry 0 rz 0 deg; joints [-3.716, -65.888, 153.382, -3.726, -86.629, 0.435]
  MoveC 754 to (267.87, -423.31, -8.35) mm, rotated rx -180 ry 0 rz 0 deg; joints [-3.745, -65.883, 153.366, -3.755, -86.62, 0.437] to (267.42, -423.49, -8.35) mm, rotated rx 180 ry 0 rz 0 deg; joints [-3.755, -65.87, 153.333, -3.765, -86.599, 0.439]
  MoveL 755 to (266.79, -423.49, -8.35) mm, rotated rx 180 ry 0 rz 0 deg; joints [-3.752, -65.854, 153.288, -3.763, -86.57, 0.441]
  MoveC 756 to (266.34, -423.49, -8.16) mm, rotated rx 180 ry 0 rz 0 deg; joints [-3.75, -65.862, 153.257, -3.761, -86.53, 0.443] to (266.15, -423.49, -7.72) mm, rotated rx 180 ry 0 rz 0 deg; joints [-3.75, -65.907, 153.245, -3.76, -86.474, 0.447]
  Set speed (500.0 mm/s)
  MoveL 757 to (266.15, -423.49, 6) mm, rotated rx 180 ry 0 rz 0 deg; joints [-3.753, -67.403, 153.285, -3.771, -85.02, 0.543]
  MoveL 758 to (139.15, -422.22, 6) mm, rotated rx -180 ry 0 rz 0 deg; joints [-3.207, -63.48, 144.059, -3.263, -79.724, 0.806]
  Set speed (25.4 mm/s)
  MoveL 759 to (139.15, -422.22, -3.54) mm, rotated rx 180 ry 0 rz 0 deg; joints [-3.205, -62.64, 144.038, -3.253, -80.543, 0.759]
  MoveC 760 to (139.34, -422.22, -3.99) mm, rotated rx -180 ry 0 rz 0 deg; joints [-3.206, -62.606, 144.051, -3.253, -80.589, 0.756] to (139.79, -422.22, -4.17) mm, rotated rx 180 ry 0 rz 0 deg; joints [-3.207, -62.603, 144.083, -3.254, -80.624, 0.754]
  Set speed (50.8 mm/s)
  MoveL 761 to (140.42, -422.22, -4.17) mm, rotated rx 180 ry 0 rz 0 deg; joints [-3.209, -62.623, 144.13, -3.256, -80.651, 0.753]
  MoveC 762 to (140.87, -422.41, -4.18) mm, rotated rx -180 ry 0 rz 0 deg; joints [-3.221, -62.637, 144.163, -3.268, -80.67, 0.754] to (141.06, -422.86, -4.18) mm, rotated rx 180 ry 0 rz 0 deg; joints [-3.247, -62.641, 144.175, -3.295, -80.677, 0.757]
  MoveL 763 to (141.06, -448.26, -4.17) mm, rotated rx -180 ry 0 rz 0 deg; joints [-4.691, -62.578, 144.044, -4.758, -80.625, 0.978]
  MoveL 764 to (90.26, -448.26, -4.18) mm, rotated rx 180 ry 0 rz 0 deg; joints [-4.466, -60.965, 140.272, -4.561, -78.47, 1.118]
  MoveL 765 to (90.26, -397.46, -4.17) mm, rotated rx 180 ry 0 rz 0 deg; joints [-1.713, -61.071, 140.479, -1.751, -78.543, 0.594]
  MoveL 766 to (141.06, -397.46, -4.18) mm, rotated rx 180 ry 0 rz 0 deg; joints [-1.799, -62.686, 144.258, -1.827, -80.707, 0.54]
  MoveL 767 to (141.06, -422.86, -4.18) mm, rotated rx 180 ry 0 rz 0 deg; joints [-3.247, -62.641, 144.175, -3.295, -80.677, 0.757]
  MoveC 768 to (140.87, -423.31, -4.18) mm, rotated rx -180 ry 0 rz 0 deg; joints [-3.272, -62.635, 144.159, -3.32, -80.669, 0.761] to (140.42, -423.49, -4.17) mm, rotated rx 180 ry 0 rz 0 deg; joints [-3.281, -62.62, 144.125, -3.329, -80.649, 0.764]
  MoveL 769 to (139.79, -423.49, -4.18) mm, rotated rx 180 ry 0 rz 0 deg; joints [-3.279, -62.601, 144.078, -3.328, -80.622, 0.765]
  MoveC 770 to (139.34, -423.49, -3.99) mm, rotated rx 180 ry 0 rz 0 deg; joints [-3.278, -62.603, 144.046, -3.326, -80.587, 0.767] to (139.15, -423.49, -3.54) mm, rotated rx -180 ry 0 rz 0 deg; joints [-3.277, -62.637, 144.033, -3.326, -80.541, 0.77]
  Set speed (500.0 mm/s)
  MoveL 771 to (139.15, -423.49, 5) mm, rotated rx 180 ry 0 rz 0 deg; joints [-3.279, -63.39, 144.052, -3.336, -79.808, 0.813]
  MoveL 772 to (139.15, -422.22, 5) mm, rotated rx -180 ry 0 rz 0 deg; joints [-3.207, -63.392, 144.057, -3.262, -79.81, 0.801]
  Set speed (25.4 mm/s)
  MoveL 773 to (139.15, -422.22, 1.82) mm, rotated rx 180 ry 0 rz 0 deg; joints [-3.206, -63.113, 144.051, -3.259, -80.083, 0.785]
  MoveL 774 to (139.15, -422.22, -7.72) mm, rotated rx -180 ry 0 rz 0 deg; joints [-3.204, -62.27, 144.026, -3.249, -80.899, 0.738]
  MoveC 775 to (139.34, -422.22, -8.16) mm, rotated rx 180 ry 0 rz 0 deg; joints [-3.205, -62.236, 144.038, -3.249, -80.945, 0.735] to (139.79, -422.22, -8.35) mm, rotated rx -180 ry 0 rz 0 deg; joints [-3.206, -62.234, 144.071, -3.25, -80.981, 0.734]
  Set speed (50.8 mm/s)
  MoveL 776 to (140.42, -422.22, -8.35) mm, rotated rx -180 ry 0 rz 0 deg; joints [-3.208, -62.253, 144.118, -3.252, -81.008, 0.732]
  MoveC 777 to (140.87, -422.41, -8.35) mm, rotated rx -180 ry 0 rz 0 deg; joints [-3.22, -62.266, 144.15, -3.264, -81.027, 0.733] to (141.06, -422.86, -8.35) mm, rotated rx 180 ry 0 rz 0 deg; joints [-3.246, -62.271, 144.162, -3.29, -81.034, 0.736]
  MoveL 778 to (141.06, -448.26, -8.35) mm, rotated rx -180 ry 0 rz 0 deg; joints [-4.69, -62.209, 144.032, -4.753, -80.981, 0.948]
  MoveL 779 to (90.26, -448.26, -8.35) mm, rotated rx -180 ry 0 rz 0 deg; joints [-4.465, -60.622, 140.26, -4.555, -78.801, 1.091]
  MoveL 780 to (90.26, -397.46, -8.35) mm, rotated rx 180 ry 0 rz 0 deg; joints [-1.712, -60.726, 140.467, -1.748, -78.875, 0.584]
  MoveL 781 to (141.06, -397.46, -8.35) mm, rotated rx 180 ry 0 rz 0 deg; joints [-1.798, -62.315, 144.245, -1.825, -81.065, 0.528]
  MoveL 782 to (141.06, -422.86, -8.35) mm, rotated rx 180 ry 0 rz 0 deg; joints [-3.246, -62.271, 144.162, -3.29, -81.034, 0.736]
  MoveC 783 to (140.87, -423.31, -8.35) mm, rotated rx -180 ry 0 rz 0 deg; joints [-3.271, -62.264, 144.146, -3.316, -81.026, 0.74] to (140.42, -423.49, -8.35) mm, rotated rx 180 ry 0 rz 0 deg; joints [-3.28, -62.25, 144.112, -3.325, -81.006, 0.743]
  MoveL 784 to (139.79, -423.49, -8.35) mm, rotated rx -180 ry 0 rz 0 deg; joints [-3.278, -62.231, 144.066, -3.323, -80.979, 0.744]
  MoveC 785 to (139.34, -423.49, -8.16) mm, rotated rx 180 ry 0 rz 0 deg; joints [-3.277, -62.234, 144.033, -3.322, -80.943, 0.746] to (139.15, -423.49, -7.72) mm, rotated rx 180 ry 0 rz 0 deg; joints [-3.276, -62.268, 144.021, -3.322, -80.897, 0.749]
  Set speed (500.0 mm/s)
  MoveL 786 to (139.15, -423.49, 6) mm, rotated rx -180 ry 0 rz 0 deg; joints [-3.279, -63.478, 144.054, -3.337, -79.722, 0.818]
  MoveL 787 to (-92.16, -422.22, 6) mm, rotated rx -180 ry 0 rz 0 deg; joints [-2.608, -55.381, 126.316, -2.778, -70.086, 1.179]
  Set speed (25.4 mm/s)
  MoveL 788 to (-92.16, -422.22, -3.54) mm, rotated rx 180 ry 0 rz 0 deg; joints [-2.606, -54.758, 126.299, -2.765, -70.692, 1.148]
  MoveC 789 to (-91.98, -422.22, -3.99) mm, rotated rx 180 ry 0 rz 0 deg; joints [-2.606, -54.735, 126.313, -2.765, -70.728, 1.146] to (-91.53, -422.22, -4.17) mm, rotated rx -180 ry 0 rz 0 deg; joints [-2.607, -54.74, 126.349, -2.765, -70.759, 1.145]
  Set speed (50.8 mm/s)
  MoveL 790 to (-90.89, -422.22, -4.18) mm, rotated rx 180 ry 0 rz 0 deg; joints [-2.608, -54.763, 126.4, -2.766, -70.787, 1.144]
  MoveC 791 to (-90.44, -422.41, -4.18) mm, rotated rx 180 ry 0 rz 0 deg; joints [-2.618, -54.779, 126.435, -2.776, -70.806, 1.146] to (-90.26, -422.86, -4.17) mm, rotated rx -180 ry 0 rz 0 deg; joints [-2.639, -54.785, 126.448, -2.798, -70.814, 1.153]
  MoveL 792 to (-90.26, -448.26, -4.17) mm, rotated rx 180 ry 0 rz 0 deg; joints [-3.814, -54.726, 126.333, -4.044, -70.78, 1.547]
  MoveL 793 to (-141.06, -448.26, -4.18) mm, rotated rx 180 ry 0 rz 0 deg; joints [-3.664, -52.83, 122.223, -3.94, -68.569, 1.658]
  MoveL 794 to (-141.06, -397.46, -4.17) mm, rotated rx -180 ry 0 rz 0 deg; joints [-1.404, -52.928, 122.408, -1.512, -68.617, 0.802]
  MoveL 795 to (-90.26, -397.46, -4.17) mm, rotated rx 180 ry 0 rz 0 deg; joints [-1.462, -54.826, 126.521, -1.552, -70.832, 0.76]
  MoveL 796 to (-90.26, -422.86, -4.17) mm, rotated rx -180 ry 0 rz 0 deg; joints [-2.639, -54.785, 126.448, -2.798, -70.814, 1.153]
  MoveC 797 to (-90.44, -423.31, -4.18) mm, rotated rx -180 ry 0 rz 0 deg; joints [-2.659, -54.777, 126.432, -2.82, -70.805, 1.16] to (-90.89, -423.49, -4.18) mm, rotated rx -180 ry 0 rz 0 deg; joints [-2.667, -54.761, 126.395, -2.829, -70.786, 1.163]
  MoveL 798 to (-91.53, -423.49, -4.17) mm, rotated rx 180 ry 0 rz 0 deg; joints [-2.666, -54.737, 126.344, -2.828, -70.758, 1.164]
  MoveC 799 to (-91.98, -423.49, -3.99) mm, rotated rx 180 ry 0 rz 0 deg; joints [-2.665, -54.733, 126.309, -2.827, -70.727, 1.166] to (-92.16, -423.49, -3.54) mm, rotated rx -180 ry 0 rz 0 deg; joints [-2.664, -54.756, 126.295, -2.827, -70.69, 1.167]
  Set speed (500.0 mm/s)
  MoveL 800 to (-92.16, -423.49, 5) mm, rotated rx 180 ry 0 rz 0 deg; joints [-2.666, -55.314, 126.31, -2.839, -70.148, 1.196]
  MoveL 801 to (-92.16, -422.22, 5) mm, rotated rx 180 ry 0 rz 0 deg; joints [-2.607, -55.316, 126.315, -2.776, -70.15, 1.176]
  Set speed (25.4 mm/s)
  MoveL 802 to (-92.16, -422.22, 1.83) mm, rotated rx 180 ry 0 rz 0 deg; joints [-2.607, -55.109, 126.31, -2.772, -70.352, 1.165]
  MoveL 803 to (-92.16, -422.22, -7.72) mm, rotated rx -180 ry 0 rz 0 deg; joints [-2.605, -54.484, 126.29, -2.76, -70.955, 1.134]
  MoveC 804 to (-91.98, -422.22, -8.16) mm, rotated rx 180 ry 0 rz 0 deg; joints [-2.605, -54.461, 126.303, -2.76, -70.992, 1.132] to (-91.53, -422.22, -8.35) mm, rotated rx -180 ry 0 rz 0 deg; joints [-2.606, -54.466, 126.339, -2.76, -71.023, 1.131]
  Set speed (50.8 mm/s)
  MoveL 805 to (-90.89, -422.22, -8.35) mm, rotated rx -180 ry 0 rz 0 deg; joints [-2.608, -54.489, 126.39, -2.761, -71.051, 1.13]
  MoveC 806 to (-90.44, -422.41, -8.35) mm, rotated rx 180 ry 0 rz 0 deg; joints [-2.617, -54.505, 126.425, -2.771, -71.07, 1.132] to (-90.26, -422.86, -8.35) mm, rotated rx 180 ry 0 rz 0 deg; joints [-2.638, -54.511, 126.438, -2.793, -71.078, 1.139]
  MoveL 807 to (-90.26, -448.26, -8.35) mm, rotated rx 180 ry 0 rz 0 deg; joints [-3.813, -54.452, 126.323, -4.036, -71.043, 1.527]
  MoveL 808 to (-141.06, -448.26, -8.35) mm, rotated rx -180 ry 0 rz 0 deg; joints [-3.663, -52.57, 122.214, -3.933, -68.818, 1.64]
  MoveL 809 to (-141.06, -397.46, -8.35) mm, rotated rx 180 ry 0 rz 0 deg; joints [-1.403, -52.668, 122.398, -1.508, -68.867, 0.795]
  MoveL 810 to (-90.26, -397.46, -8.35) mm, rotated rx -180 ry 0 rz 0 deg; joints [-1.461, -54.551, 126.511, -1.548, -71.097, 0.752]
  MoveL 811 to (-90.26, -422.86, -8.35) mm, rotated rx 180 ry 0 rz 0 deg; joints [-2.638, -54.511, 126.438, -2.793, -71.078, 1.139]
  MoveC 812 to (-90.44, -423.31, -8.35) mm, rotated rx -180 ry 0 rz 0 deg; joints [-2.659, -54.503, 126.422, -2.815, -71.069, 1.146] to (-90.89, -423.49, -8.35) mm, rotated rx 180 ry 0 rz 0 deg; joints [-2.666, -54.486, 126.385, -2.823, -71.05, 1.149]
  MoveL 813 to (-91.53, -423.49, -8.35) mm, rotated rx -180 ry 0 rz 0 deg; joints [-2.665, -54.463, 126.334, -2.822, -71.022, 1.15]
  MoveC 814 to (-91.98, -423.49, -8.16) mm, rotated rx -180 ry 0 rz 0 deg; joints [-2.664, -54.459, 126.299, -2.822, -70.991, 1.152] to (-92.16, -423.49, -7.72) mm, rotated rx -180 ry 0 rz 0 deg; joints [-2.664, -54.482, 126.285, -2.822, -70.954, 1.153]
  Set speed (500.0 mm/s)
  MoveL 815 to (-92.16, -423.49, 6) mm, rotated rx 180 ry 0 rz 0 deg; joints [-2.666, -55.379, 126.311, -2.84, -70.085, 1.2]
  MoveL 816 to (-219.16, -422.22, 6) mm, rotated rx -180 ry 0 rz 0 deg; joints [-2.365, -50.425, 115.83, -2.623, -64.558, 1.364]
  Set speed (25.4 mm/s)
  MoveL 817 to (-219.16, -422.22, -3.54) mm, rotated rx -180 ry 0 rz 0 deg; joints [-2.363, -49.879, 115.814, -2.61, -65.087, 1.336]
  MoveC 818 to (-218.98, -422.22, -3.99) mm, rotated rx -180 ry 0 rz 0 deg; joints [-2.363, -49.861, 115.829, -2.609, -65.121, 1.335] to (-218.53, -422.22, -4.17) mm, rotated rx -180 ry 0 rz 0 deg; joints [-2.364, -49.868, 115.867, -2.61, -65.151, 1.334]
  Set speed (50.8 mm/s)
  MoveL 819 to (-217.89, -422.22, -4.18) mm, rotated rx -180 ry 0 rz 0 deg; joints [-2.365, -49.894, 115.921, -2.61, -65.18, 1.333]
  MoveC 820 to (-217.44, -422.41, -4.18) mm, rotated rx -180 ry 0 rz 0 deg; joints [-2.374, -49.911, 115.959, -2.619, -65.2, 1.335] to (-217.26, -422.86, -4.17) mm, rotated rx 180 ry 0 rz 0 deg; joints [-2.393, -49.918, 115.973, -2.64, -65.208, 1.344]
  MoveL 821 to (-217.26, -448.26, -4.18) mm, rotated rx -180 ry 0 rz 0 deg; joints [-3.459, -49.86, 115.862, -3.816, -65.179, 1.823]
  MoveL 822 to (-268.06, -448.26, -4.17) mm, rotated rx 180 ry 0 rz 0 deg; joints [-3.335, -47.79, 111.469, -3.752, -62.858, 1.935]
  MoveL 823 to (-268.06, -397.46, -4.18) mm, rotated rx 180 ry 0 rz 0 deg; joints [-1.277, -47.886, 111.65, -1.439, -62.901, 0.909]
  MoveL 824 to (-217.26, -397.46, -4.18) mm, rotated rx 180 ry 0 rz 0 deg; joints [-1.325, -49.957, 116.044, -1.464, -65.224, 0.866]
  MoveL 825 to (-217.26, -422.86, -4.17) mm, rotated rx 180 ry 0 rz 0 deg; joints [-2.393, -49.918, 115.973, -2.64, -65.208, 1.344]
  MoveC 826 to (-217.44, -423.31, -4.17) mm, rotated rx -180 ry 0 rz 0 deg; joints [-2.411, -49.91, 115.956, -2.661, -65.199, 1.352] to (-217.89, -423.49, -4.18) mm, rotated rx 180 ry 0 rz 0 deg; joints [-2.418, -49.891, 115.917, -2.669, -65.179, 1.357]
  MoveL 827 to (-218.53, -423.49, -4.18) mm, rotated rx -180 ry 0 rz 0 deg; joints [-2.417, -49.866, 115.863, -2.668, -65.15, 1.358]
  MoveC 828 to (-218.98, -423.49, -3.99) mm, rotated rx -180 ry 0 rz 0 deg; joints [-2.416, -49.859, 115.825, -2.668, -65.12, 1.359] to (-219.16, -423.49, -3.54) mm, rotated rx -180 ry 0 rz 0 deg; joints [-2.416, -49.877, 115.81, -2.669, -65.086, 1.36]
  Set speed (500.0 mm/s)
  MoveL 829 to (-219.16, -423.49, 5) mm, rotated rx 180 ry 0 rz 0 deg; joints [-2.418, -50.366, 115.824, -2.681, -64.612, 1.386]
  MoveL 830 to (-219.16, -422.22, 5) mm, rotated rx -180 ry 0 rz 0 deg; joints [-2.364, -50.368, 115.829, -2.622, -64.613, 1.361]
  Set speed (25.4 mm/s)
  MoveL 831 to (-219.16, -422.22, 1.83) mm, rotated rx 180 ry 0 rz 0 deg; joints [-2.364, -50.187, 115.824, -2.617, -64.79, 1.352]
  MoveL 832 to (-219.16, -422.22, -7.72) mm, rotated rx 180 ry 0 rz 0 deg; joints [-2.362, -49.639, 115.805, -2.604, -65.318, 1.324]
  MoveC 833 to (-218.98, -422.22, -8.16) mm, rotated rx -180 ry 0 rz 0 deg; joints [-2.362, -49.621, 115.82, -2.604, -65.351, 1.323] to (-218.53, -422.22, -8.35) mm, rotated rx -180 ry 0 rz 0 deg; joints [-2.363, -49.628, 115.858, -2.604, -65.382, 1.322]
  Set speed (50.8 mm/s)
  MoveL 834 to (-217.89, -422.22, -8.35) mm, rotated rx -180 ry 0 rz 0 deg; joints [-2.364, -49.653, 115.912, -2.605, -65.411, 1.321]
  MoveC 835 to (-217.44, -422.41, -8.35) mm, rotated rx 180 ry 0 rz 0 deg; joints [-2.373, -49.671, 115.95, -2.614, -65.431, 1.324] to (-217.26, -422.86, -8.35) mm, rotated rx 180 ry 0 rz 0 deg; joints [-2.392, -49.677, 115.964, -2.634, -65.439, 1.332]
  MoveL 836 to (-217.26, -448.26, -8.35) mm, rotated rx -180 ry 0 rz 0 deg; joints [-3.458, -49.62, 115.853, -3.808, -65.41, 1.806]
  MoveL 837 to (-268.06, -448.26, -8.35) mm, rotated rx -180 ry 0 rz 0 deg; joints [-3.334, -47.561, 111.46, -3.744, -63.078, 1.919]
  MoveL 838 to (-268.06, -397.46, -8.35) mm, rotated rx 180 ry 0 rz 0 deg; joints [-1.277, -47.657, 111.64, -1.436, -63.121, 0.902]
  MoveL 839 to (-217.26, -397.46, -8.35) mm, rotated rx 180 ry 0 rz 0 deg; joints [-1.324, -49.717, 116.034, -1.46, -65.455, 0.859]
  MoveL 840 to (-217.26, -422.86, -8.35) mm, rotated rx 180 ry 0 rz 0 deg; joints [-2.392, -49.677, 115.964, -2.634, -65.439, 1.332]
  MoveC 841 to (-217.44, -423.31, -8.35) mm, rotated rx -180 ry 0 rz 0 deg; joints [-2.411, -49.669, 115.946, -2.655, -65.43, 1.34] to (-217.89, -423.49, -8.35) mm, rotated rx -180 ry 0 rz 0 deg; joints [-2.418, -49.651, 115.907, -2.663, -65.41, 1.344]
  MoveL 842 to (-218.53, -423.49, -8.35) mm, rotated rx -180 ry 0 rz 0 deg; joints [-2.417, -49.626, 115.853, -2.663, -65.381, 1.345]
  MoveC 843 to (-218.98, -423.49, -8.16) mm, rotated rx 180 ry 0 rz 0 deg; joints [-2.416, -49.618, 115.815, -2.662, -65.35, 1.347] to (-219.16, -423.49, -7.72) mm, rotated rx -180 ry 0 rz 0 deg; joints [-2.416, -49.637, 115.801, -2.663, -65.317, 1.348]
  Set speed (500.0 mm/s)
  MoveL 844 to (-219.16, -423.49, 6) mm, rotated rx 180 ry 0 rz 0 deg; joints [-2.418, -50.423, 115.825, -2.682, -64.557, 1.389]
  MoveL 845 to (-346.16, -422.22, 6) mm, rotated rx 180 ry 0 rz 0 deg; joints [-2.163, -45.022, 104.557, -2.536, -58.69, 1.558]
  Set speed (25.4 mm/s)
  MoveL 846 to (-346.16, -422.22, -3.54) mm, rotated rx -180 ry 0 rz 0 deg; joints [-2.161, -44.536, 104.542, -2.522, -59.16, 1.533]
  MoveC 847 to (-345.98, -422.22, -3.99) mm, rotated rx 180 ry 0 rz 0 deg; joints [-2.162, -44.521, 104.558, -2.522, -59.191, 1.532] to (-345.53, -422.22, -4.17) mm, rotated rx -180 ry 0 rz 0 deg; joints [-2.162, -44.532, 104.599, -2.521, -59.222, 1.53]
  Set speed (50.8 mm/s)
  MoveL 848 to (-344.89, -422.22, -4.18) mm, rotated rx -180 ry 0 rz 0 deg; joints [-2.163, -44.56, 104.658, -2.522, -59.253, 1.529]
  MoveC 849 to (-344.44, -422.41, -4.18) mm, rotated rx -180 ry 0 rz 0 deg; joints [-2.171, -44.579, 104.699, -2.53, -59.274, 1.533] to (-344.26, -422.86, -4.18) mm, rotated rx 180 ry 0 rz 0 deg; joints [-2.189, -44.586, 104.715, -2.55, -59.283, 1.542]
  MoveL 850 to (-344.26, -448.26, -4.18) mm, rotated rx -180 ry 0 rz 0 deg; joints [-3.164, -44.529, 104.605, -3.687, -59.257, 2.111]
  MoveL 851 to (-395.06, -448.26, -4.17) mm, rotated rx 180 ry 0 rz 0 deg; joints [-3.06, -42.236, 99.81, -3.664, -56.757, 2.236]
  MoveL 852 to (-395.06, -397.46, -4.17) mm, rotated rx -180 ry 0 rz 0 deg; joints [-1.172, -42.333, 99.991, -1.405, -56.796, 1.024]
  MoveL 853 to (-344.26, -397.46, -4.17) mm, rotated rx -180 ry 0 rz 0 deg; joints [-1.212, -44.625, 104.785, -1.414, -59.297, 0.976]
  MoveL 854 to (-344.26, -422.86, -4.18) mm, rotated rx 180 ry 0 rz 0 deg; joints [-2.189, -44.586, 104.715, -2.55, -59.283, 1.542]
  MoveC 855 to (-344.44, -423.31, -4.18) mm, rotated rx -180 ry 0 rz 0 deg; joints [-2.206, -44.577, 104.696, -2.57, -59.274, 1.553] to (-344.89, -423.49, -4.18) mm, rotated rx 180 ry 0 rz 0 deg; joints [-2.212, -44.557, 104.654, -2.579, -59.252, 1.558]
  MoveL 856 to (-345.53, -423.49, -4.18) mm, rotated rx -180 ry 0 rz 0 deg; joints [-2.211, -44.529, 104.595, -2.578, -59.221, 1.559]
  MoveC 857 to (-345.98, -423.49, -3.99) mm, rotated rx -180 ry 0 rz 0 deg; joints [-2.21, -44.519, 104.554, -2.578, -59.19, 1.56] to (-346.16, -423.49, -3.54) mm, rotated rx -180 ry 0 rz 0 deg; joints [-2.21, -44.534, 104.537, -2.579, -59.159, 1.562]
  Set speed (500.0 mm/s)
  MoveL 858 to (-346.16, -423.49, 5) mm, rotated rx -180 ry 0 rz 0 deg; joints [-2.212, -44.969, 104.551, -2.592, -58.738, 1.584]
  MoveL 859 to (-346.16, -422.22, 5) mm, rotated rx 180 ry 0 rz 0 deg; joints [-2.163, -44.971, 104.556, -2.535, -58.739, 1.556]
  Set speed (25.4 mm/s)
  MoveL 860 to (-346.16, -422.22, 1.83) mm, rotated rx -180 ry 0 rz 0 deg; joints [-2.162, -44.81, 104.551, -2.53, -58.896, 1.547]
  MoveL 861 to (-346.16, -422.22, -7.71) mm, rotated rx -180 ry 0 rz 0 deg; joints [-2.161, -44.322, 104.533, -2.516, -59.365, 1.522]
  MoveC 862 to (-345.98, -422.22, -8.16) mm, rotated rx -180 ry 0 rz 0 deg; joints [-2.161, -44.307, 104.549, -2.515, -59.396, 1.521] to (-345.53, -422.22, -8.35) mm, rotated rx -180 ry 0 rz 0 deg; joints [-2.162, -44.318, 104.59, -2.515, -59.427, 1.519]
  Set speed (50.8 mm/s)
  MoveL 863 to (-344.89, -422.22, -8.35) mm, rotated rx -180 ry 0 rz 0 deg; joints [-2.163, -44.346, 104.649, -2.516, -59.458, 1.518]
  MoveC 864 to (-344.44, -422.41, -8.35) mm, rotated rx -180 ry 0 rz 0 deg; joints [-2.17, -44.365, 104.69, -2.524, -59.479, 1.522] to (-344.26, -422.86, -8.35) mm, rotated rx 180 ry 0 rz 0 deg; joints [-2.188, -44.372, 104.706, -2.544, -59.488, 1.531]
  MoveL 865 to (-344.26, -448.26, -8.35) mm, rotated rx 180 ry 0 rz 0 deg; joints [-3.164, -44.315, 104.595, -3.678, -59.462, 2.095]
  MoveL 866 to (-395.06, -448.26, -8.35) mm, rotated rx -180 ry 0 rz 0 deg; joints [-3.059, -42.031, 99.801, -3.655, -56.953, 2.221]
  MoveL 867 to (-395.06, -397.46, -8.35) mm, rotated rx 180 ry 0 rz 0 deg; joints [-1.171, -42.128, 99.982, -1.401, -56.993, 1.018]
  MoveL 868 to (-344.26, -397.46, -8.35) mm, rotated rx -180 ry 0 rz 0 deg; joints [-1.211, -44.411, 104.776, -1.41, -59.503, 0.97]
  MoveL 869 to (-344.26, -422.86, -8.35) mm, rotated rx 180 ry 0 rz 0 deg; joints [-2.188, -44.372, 104.706, -2.544, -59.488, 1.531]
  MoveC 870 to (-344.44, -423.31, -8.35) mm, rotated rx 180 ry 0 rz 0 deg; joints [-2.205, -44.363, 104.687, -2.564, -59.479, 1.542] to (-344.89, -423.49, -8.35) mm, rotated rx -180 ry 0 rz 0 deg; joints [-2.211, -44.343, 104.645, -2.572, -59.457, 1.547]
  MoveL 871 to (-345.53, -423.49, -8.35) mm, rotated rx -180 ry 0 rz 0 deg; joints [-2.21, -44.315, 104.586, -2.572, -59.426, 1.548]
  MoveC 872 to (-345.98, -423.49, -8.16) mm, rotated rx 180 ry 0 rz 0 deg; joints [-2.21, -44.305, 104.545, -2.572, -59.395, 1.549] to (-346.16, -423.49, -7.72) mm, rotated rx -180 ry 0 rz 0 deg; joints [-2.21, -44.32, 104.529, -2.573, -59.364, 1.55]
  Set speed (500.0 mm/s)
  MoveL 873 to (-346.16, -423.49, 6) mm, rotated rx -180 ry 0 rz 0 deg; joints [-2.212, -45.019, 104.552, -2.594, -58.689, 1.587]
  MoveL 874 to (-346.16, -235.89, 6) mm, rotated rx 180 ry 0 rz 0 deg; joints [4.986, -44.865, 104.132, 5.844, -58.527, -2.71]
  Set speed (25.4 mm/s)
  MoveL 875 to (-346.16, -235.88, -3.54) mm, rotated rx -180 ry 0 rz 0 deg; joints [4.989, -44.381, 104.117, 5.817, -58.994, -2.656]
  MoveC 876 to (-345.98, -235.89, -3.99) mm, rotated rx -180 ry 0 rz 0 deg; joints [4.989, -44.366, 104.134, 5.816, -59.025, -2.653] to (-345.53, -235.89, -4.17) mm, rotated rx 180 ry 0 rz 0 deg; joints [4.991, -44.377, 104.175, 5.816, -59.056, -2.65]
  Set speed (50.8 mm/s)
  MoveL 877 to (-344.89, -235.89, -4.18) mm, rotated rx -180 ry 0 rz 0 deg; joints [4.993, -44.405, 104.234, 5.817, -59.087, -2.648]
  MoveC 878 to (-344.44, -236.07, -4.17) mm, rotated rx -180 ry 0 rz 0 deg; joints [4.987, -44.425, 104.277, 5.809, -59.109, -2.642] to (-344.26, -236.52, -4.18) mm, rotated rx -180 ry 0 rz 0 deg; joints [4.971, -44.435, 104.298, 5.789, -59.119, -2.631]
  MoveL 879 to (-344.26, -261.92, -4.18) mm, rotated rx -180 ry 0 rz 0 deg; joints [3.999, -44.515, 104.481, 4.653, -59.178, -2.055]
  MoveL 880 to (-395.06, -261.92, -4.18) mm, rotated rx -180 ry 0 rz 0 deg; joints [3.868, -42.22, 99.686, 4.624, -56.68, -2.213]
  MoveL 881 to (-395.06, -211.12, -4.18) mm, rotated rx -180 ry 0 rz 0 deg; joints [5.745, -42.037, 99.275, 6.885, -56.555, -3.447]
  MoveL 882 to (-344.26, -211.12, -4.18) mm, rotated rx 180 ry 0 rz 0 deg; joints [5.94, -44.336, 104.074, 6.925, -59.049, -3.212]
  MoveL 883 to (-344.26, -236.52, -4.18) mm, rotated rx -180 ry 0 rz 0 deg; joints [4.971, -44.435, 104.298, 5.789, -59.119, -2.631]
  MoveC 884 to (-344.44, -236.97, -4.18) mm, rotated rx -180 ry 0 rz 0 deg; joints [4.953, -44.428, 104.284, 5.769, -59.111, -2.621] to (-344.89, -237.16, -4.18) mm, rotated rx -180 ry 0 rz 0 deg; joints [4.944, -44.409, 104.244, 5.76, -59.09, -2.619]
  MoveL 885 to (-345.53, -237.16, -4.18) mm, rotated rx -180 ry 0 rz 0 deg; joints [4.942, -44.381, 104.185, 5.759, -59.059, -2.621]
  MoveC 886 to (-345.98, -237.16, -3.99) mm, rotated rx -180 ry 0 rz 0 deg; joints [4.941, -44.371, 104.144, 5.76, -59.028, -2.624] to (-346.16, -237.16, -3.54) mm, rotated rx -180 ry 0 rz 0 deg; joints [4.94, -44.385, 104.127, 5.761, -58.997, -2.627]
  Set speed (500.0 mm/s)
  MoveL 887 to (-346.16, -237.16, 5) mm, rotated rx 180 ry 0 rz 0 deg; joints [4.938, -44.819, 104.141, 5.784, -58.58, -2.675]
  MoveL 888 to (-346.16, -235.89, 5) mm, rotated rx 180 ry 0 rz 0 deg; joints [4.987, -44.814, 104.131, 5.841, -58.577, -2.705]
  Set speed (25.4 mm/s)
  MoveL 889 to (-346.16, -235.89, 1.83) mm, rotated rx 180 ry 0 rz 0 deg; joints [4.987, -44.653, 104.126, 5.832, -58.732, -2.687]
  MoveL 890 to (-346.16, -235.88, -7.71) mm, rotated rx -180 ry 0 rz 0 deg; joints [4.99, -44.168, 104.108, 5.806, -59.197, -2.633]
  MoveC 891 to (-345.98, -235.89, -8.16) mm, rotated rx -180 ry 0 rz 0 deg; joints [4.99, -44.153, 104.125, 5.805, -59.228, -2.629] to (-345.53, -235.89, -8.35) mm, rotated rx 180 ry 0 rz 0 deg; joints [4.992, -44.164, 104.166, 5.805, -59.259, -2.627]
  Set speed (50.8 mm/s)
  MoveL 892 to (-344.89, -235.89, -8.35) mm, rotated rx 180 ry 0 rz 0 deg; joints [4.994, -44.192, 104.225, 5.806, -59.29, -2.624]
  MoveC 893 to (-344.44, -236.07, -8.35) mm, rotated rx -180 ry 0 rz 0 deg; joints [4.988, -44.212, 104.268, 5.798, -59.312, -2.618] to (-344.26, -236.52, -8.35) mm, rotated rx 180 ry 0 rz 0 deg; joints [4.972, -44.222, 104.289, 5.778, -59.322, -2.607]
  MoveL 894 to (-344.26, -261.92, -8.35) mm, rotated rx -180 ry 0 rz 0 deg; joints [4, -44.302, 104.472, 4.644, -59.382, -2.036]
  MoveL 895 to (-395.06, -261.92, -8.35) mm, rotated rx -180 ry 0 rz 0 deg; joints [3.869, -42.015, 99.677, 4.615, -56.875, -2.195]
  MoveL 896 to (-395.06, -211.12, -8.35) mm, rotated rx -180 ry 0 rz 0 deg; joints [5.746, -41.833, 99.266, 6.87, -56.748, -3.42]
  MoveL 897 to (-344.26, -211.12, -8.35) mm, rotated rx -180 ry 0 rz 0 deg; joints [5.941, -44.123, 104.065, 6.911, -59.251, -3.184]
  MoveL 898 to (-344.26, -236.52, -8.35) mm, rotated rx 180 ry 0 rz 0 deg; joints [4.972, -44.222, 104.289, 5.778, -59.322, -2.607]
  MoveC 899 to (-344.44, -236.97, -8.35) mm, rotated rx -180 ry 0 rz 0 deg; joints [4.954, -44.215, 104.275, 5.758, -59.314, -2.598] to (-344.89, -237.16, -8.35) mm, rotated rx -180 ry 0 rz 0 deg; joints [4.945, -44.196, 104.235, 5.749, -59.293, -2.595]
  MoveL 900 to (-345.53, -237.16, -8.35) mm, rotated rx 180 ry 0 rz 0 deg; joints [4.943, -44.168, 104.176, 5.748, -59.262, -2.598]
  MoveC 901 to (-345.98, -237.15, -8.16) mm, rotated rx -180 ry 0 rz 0 deg; joints [4.942, -44.158, 104.135, 5.748, -59.231, -2.601] to (-346.16, -237.16, -7.72) mm, rotated rx -180 ry 0 rz 0 deg; joints [4.941, -44.173, 104.119, 5.749, -59.201, -2.604]
  Set speed (500.0 mm/s)
  MoveL 902 to (-346.16, -237.16, 6) mm, rotated rx -180 ry 0 rz 0 deg; joints [4.938, -44.869, 104.142, 5.787, -58.531, -2.681]
  MoveL 903 to (-219.16, -235.89, 6) mm, rotated rx 180 ry 0 rz 0 deg; joints [5.448, -50.276, 115.402, 6.039, -64.378, -2.264]
  Set speed (25.4 mm/s)
  MoveL 904 to (-219.16, -235.89, -3.54) mm, rotated rx 180 ry 0 rz 0 deg; joints [5.45, -49.732, 115.387, 6.015, -64.903, -2.204]
  MoveC 905 to (-218.98, -235.89, -3.99) mm, rotated rx 180 ry 0 rz 0 deg; joints [5.451, -49.714, 115.402, 6.014, -64.936, -2.2] to (-218.53, -235.89, -4.17) mm, rotated rx 180 ry 0 rz 0 deg; joints [5.453, -49.722, 115.44, 6.015, -64.966, -2.198]
  Set speed (50.8 mm/s)
  MoveL 906 to (-217.89, -235.89, -4.18) mm, rotated rx 180 ry 0 rz 0 deg; joints [5.455, -49.747, 115.494, 6.016, -64.995, -2.195]
  MoveC 907 to (-217.44, -236.07, -4.18) mm, rotated rx 180 ry 0 rz 0 deg; joints [5.449, -49.766, 115.534, 6.009, -65.016, -2.19] to (-217.26, -236.52, -4.18) mm, rotated rx -180 ry 0 rz 0 deg; joints [5.431, -49.775, 115.553, 5.988, -65.025, -2.181]
  MoveL 908 to (-217.26, -261.92, -4.17) mm, rotated rx -180 ry 0 rz 0 deg; joints [4.37, -49.853, 115.738, 4.814, -65.091, -1.693]
  MoveL 909 to (-268.06, -261.92, -4.18) mm, rotated rx -180 ry 0 rz 0 deg; joints [4.214, -47.78, 111.346, 4.735, -62.774, -1.834]
  MoveL 910 to (-268.06, -211.12, -4.18) mm, rotated rx -180 ry 0 rz 0 deg; joints [6.257, -47.604, 110.938, 7.044, -62.637, -2.883]
  MoveL 911 to (-217.26, -211.12, -4.17) mm, rotated rx -180 ry 0 rz 0 deg; joints [6.489, -49.678, 115.328, 7.161, -64.948, -2.674]
  MoveL 912 to (-217.26, -236.52, -4.18) mm, rotated rx -180 ry 0 rz 0 deg; joints [5.431, -49.775, 115.553, 5.988, -65.025, -2.181]
  MoveC 913 to (-217.44, -236.97, -4.18) mm, rotated rx -180 ry 0 rz 0 deg; joints [5.412, -49.769, 115.541, 5.967, -65.018, -2.173] to (-217.89, -237.15, -4.18) mm, rotated rx 180 ry 0 rz 0 deg; joints [5.402, -49.752, 115.504, 5.958, -64.999, -2.171]
  MoveL 914 to (-218.53, -237.16, -4.18) mm, rotated rx 180 ry 0 rz 0 deg; joints [5.4, -49.726, 115.45, 5.956, -64.97, -2.173]
  MoveC 915 to (-218.98, -237.16, -3.99) mm, rotated rx -180 ry 0 rz 0 deg; joints [5.398, -49.719, 115.412, 5.956, -64.94, -2.176] to (-219.16, -237.16, -3.54) mm, rotated rx -180 ry 0 rz 0 deg; joints [5.397, -49.737, 115.398, 5.956, -64.907, -2.179]
  Set speed (500.0 mm/s)
  MoveL 916 to (-219.16, -237.16, 5) mm, rotated rx 180 ry 0 rz 0 deg; joints [5.395, -50.223, 115.412, 5.977, -64.437, -2.232]
  MoveL 917 to (-219.16, -235.89, 5) mm, rotated rx -180 ry 0 rz 0 deg; joints [5.448, -50.219, 115.401, 6.036, -64.433, -2.258]
  Set speed (25.4 mm/s)
  MoveL 918 to (-219.16, -235.89, 1.82) mm, rotated rx 180 ry 0 rz 0 deg; joints [5.449, -50.038, 115.397, 6.028, -64.608, -2.238]
  MoveL 919 to (-219.16, -235.89, -7.72) mm, rotated rx -180 ry 0 rz 0 deg; joints [5.451, -49.494, 115.378, 6.005, -65.132, -2.178]
  MoveC 920 to (-218.98, -235.89, -8.16) mm, rotated rx 180 ry 0 rz 0 deg; joints [5.452, -49.475, 115.393, 6.004, -65.164, -2.174] to (-218.53, -235.89, -8.35) mm, rotated rx -180 ry 0 rz 0 deg; joints [5.454, -49.483, 115.431, 6.005, -65.195, -2.172]
  Set speed (50.8 mm/s)
  MoveL 921 to (-217.89, -235.88, -8.35) mm, rotated rx -180 ry 0 rz 0 deg; joints [5.456, -49.508, 115.485, 6.006, -65.224, -2.169]
  MoveC 922 to (-217.44, -236.07, -8.35) mm, rotated rx 180 ry 0 rz 0 deg; joints [5.45, -49.527, 115.525, 5.999, -65.245, -2.164] to (-217.26, -236.52, -8.35) mm, rotated rx 180 ry 0 rz 0 deg; joints [5.432, -49.535, 115.544, 5.978, -65.254, -2.155]
  MoveL 923 to (-217.26, -261.92, -8.35) mm, rotated rx -180 ry 0 rz 0 deg; joints [4.371, -49.613, 115.729, 4.807, -65.32, -1.672]
  MoveL 924 to (-268.06, -261.92, -8.35) mm, rotated rx 180 ry 0 rz 0 deg; joints [4.215, -47.552, 111.337, 4.727, -62.993, -1.814]
  MoveL 925 to (-268.06, -211.12, -8.35) mm, rotated rx 180 ry 0 rz 0 deg; joints [6.259, -47.376, 110.929, 7.031, -62.854, -2.853]
  MoveL 926 to (-217.26, -211.12, -8.35) mm, rotated rx 180 ry 0 rz 0 deg; joints [6.49, -49.439, 115.319, 7.149, -65.175, -2.643]
  MoveL 927 to (-217.26, -236.52, -8.35) mm, rotated rx 180 ry 0 rz 0 deg; joints [5.432, -49.535, 115.544, 5.978, -65.254, -2.155]
  MoveC 928 to (-217.44, -236.97, -8.35) mm, rotated rx 180 ry 0 rz 0 deg; joints [5.413, -49.53, 115.532, 5.957, -65.247, -2.147] to (-217.89, -237.15, -8.35) mm, rotated rx 180 ry 0 rz 0 deg; joints [5.403, -49.512, 115.495, 5.948, -65.227, -2.145]
  MoveL 929 to (-218.53, -237.16, -8.35) mm, rotated rx -180 ry 0 rz 0 deg; joints [5.401, -49.487, 115.441, 5.946, -65.199, -2.147]
  MoveC 930 to (-218.98, -237.16, -8.16) mm, rotated rx 180 ry 0 rz 0 deg; joints [5.399, -49.48, 115.403, 5.946, -65.168, -2.15] to (-219.16, -237.16, -7.72) mm, rotated rx 180 ry 0 rz 0 deg; joints [5.398, -49.498, 115.388, 5.947, -65.135, -2.153]
  Set speed (500.0 mm/s)
  MoveL 931 to (-219.16, -237.16, 6) mm, rotated rx -180 ry 0 rz 0 deg; joints [5.395, -50.28, 115.413, 5.98, -64.381, -2.239]
  MoveL 932 to (-92.16, -235.88, 6) mm, rotated rx -180 ry 0 rz 0 deg; joints [6.003, -55.236, 125.874, 6.389, -69.879, -1.842]
  Set speed (25.4 mm/s)
  MoveL 933 to (-92.16, -235.89, -3.54) mm, rotated rx -180 ry 0 rz 0 deg; joints [6.006, -54.617, 125.858, 6.368, -70.478, -1.772]
  MoveC 934 to (-91.98, -235.88, -3.99) mm, rotated rx -180 ry 0 rz 0 deg; joints [6.007, -54.595, 125.872, 6.368, -70.514, -1.768] to (-91.53, -235.88, -4.17) mm, rotated rx -180 ry 0 rz 0 deg; joints [6.009, -54.599, 125.907, 6.369, -70.545, -1.765]
  Set speed (50.8 mm/s)
  MoveL 935 to (-90.89, -235.89, -4.18) mm, rotated rx -180 ry 0 rz 0 deg; joints [6.012, -54.622, 125.958, 6.371, -70.573, -1.763]
  MoveC 936 to (-90.44, -236.07, -4.18) mm, rotated rx -180 ry 0 rz 0 deg; joints [6.006, -54.64, 125.995, 6.364, -70.593, -1.759] to (-90.26, -236.52, -4.18) mm, rotated rx 180 ry 0 rz 0 deg; joints [5.986, -54.648, 126.014, 6.342, -70.602, -1.751]
  MoveL 937 to (-90.26, -261.92, -4.18) mm, rotated rx -180 ry 0 rz 0 deg; joints [4.817, -54.726, 126.205, 5.101, -70.678, -1.346]
  MoveL 938 to (-141.06, -261.92, -4.17) mm, rotated rx 180 ry 0 rz 0 deg; joints [4.628, -52.827, 122.097, 4.971, -68.472, -1.485]
  MoveL 939 to (-141.06, -211.12, -4.18) mm, rotated rx -180 ry 0 rz 0 deg; joints [6.87, -52.652, 121.68, 7.39, -68.317, -2.367]
  MoveL 940 to (-90.26, -211.12, -4.18) mm, rotated rx -180 ry 0 rz 0 deg; joints [7.149, -54.551, 125.781, 7.581, -70.512, -2.161]
  MoveL 941 to (-90.26, -236.52, -4.18) mm, rotated rx 180 ry 0 rz 0 deg; joints [5.986, -54.648, 126.014, 6.342, -70.602, -1.751]
  MoveC 942 to (-90.44, -236.97, -4.17) mm, rotated rx -180 ry 0 rz 0 deg; joints [5.964, -54.643, 126.003, 6.32, -70.595, -1.744] to (-90.89, -237.16, -4.17) mm, rotated rx 180 ry 0 rz 0 deg; joints [5.954, -54.627, 125.968, 6.309, -70.577, -1.743]
  MoveL 943 to (-91.53, -237.15, -4.18) mm, rotated rx -180 ry 0 rz 0 deg; joints [5.951, -54.603, 125.918, 6.307, -70.549, -1.745]
  MoveC 944 to (-91.98, -237.16, -3.99) mm, rotated rx 180 ry 0 rz 0 deg; joints [5.948, -54.599, 125.882, 6.306, -70.518, -1.748] to (-92.16, -237.15, -3.54) mm, rotated rx -180 ry 0 rz 0 deg; joints [5.947, -54.621, 125.868, 6.306, -70.482, -1.752]
  Set speed (500.0 mm/s)
  MoveL 945 to (-92.16, -237.15, 5) mm, rotated rx -180 ry 0 rz 0 deg; joints [5.945, -55.176, 125.883, 6.325, -69.946, -1.814]
  MoveL 946 to (-92.16, -235.88, 5) mm, rotated rx -180 ry 0 rz 0 deg; joints [6.003, -55.172, 125.873, 6.387, -69.942, -1.835]
  Set speed (25.4 mm/s)
  MoveL 947 to (-92.16, -235.88, 1.82) mm, rotated rx -180 ry 0 rz 0 deg; joints [6.004, -54.966, 125.868, 6.38, -70.142, -1.811]
  MoveL 948 to (-92.16, -235.89, -7.72) mm, rotated rx 180 ry 0 rz 0 deg; joints [6.007, -54.345, 125.848, 6.359, -70.739, -1.742]
  MoveC 949 to (-91.98, -235.88, -8.16) mm, rotated rx -180 ry 0 rz 0 deg; joints [6.008, -54.322, 125.862, 6.359, -70.775, -1.738] to (-91.53, -235.88, -8.35) mm, rotated rx -180 ry 0 rz 0 deg; joints [6.01, -54.327, 125.897, 6.36, -70.806, -1.735]
  Set speed (50.8 mm/s)
  MoveL 950 to (-90.89, -235.89, -8.35) mm, rotated rx 180 ry 0 rz 0 deg; joints [6.013, -54.35, 125.948, 6.362, -70.834, -1.733]
  MoveC 951 to (-90.44, -236.07, -8.35) mm, rotated rx 180 ry 0 rz 0 deg; joints [6.007, -54.367, 125.985, 6.355, -70.854, -1.728] to (-90.26, -236.52, -8.35) mm, rotated rx -180 ry 0 rz 0 deg; joints [5.987, -54.375, 126.004, 6.334, -70.863, -1.72]
  MoveL 952 to (-90.26, -261.92, -8.35) mm, rotated rx -180 ry 0 rz 0 deg; joints [4.819, -54.452, 126.195, 5.094, -70.94, -1.322]
  MoveL 953 to (-141.06, -261.92, -8.35) mm, rotated rx -180 ry 0 rz 0 deg; joints [4.629, -52.568, 122.088, 4.964, -68.721, -1.463]
  MoveL 954 to (-141.06, -211.12, -8.35) mm, rotated rx 180 ry 0 rz 0 deg; joints [6.871, -52.394, 121.67, 7.379, -68.563, -2.333]
  MoveL 955 to (-90.26, -211.12, -8.35) mm, rotated rx -180 ry 0 rz 0 deg; joints [7.151, -54.279, 125.771, 7.57, -70.772, -2.125]
  MoveL 956 to (-90.26, -236.52, -8.35) mm, rotated rx -180 ry 0 rz 0 deg; joints [5.987, -54.375, 126.004, 6.334, -70.863, -1.72]
  MoveC 957 to (-90.44, -236.97, -8.35) mm, rotated rx 180 ry 0 rz 0 deg; joints [5.966, -54.37, 125.993, 6.311, -70.857, -1.714] to (-90.89, -237.16, -8.35) mm, rotated rx -180 ry 0 rz 0 deg; joints [5.955, -54.354, 125.958, 6.3, -70.838, -1.713]
  MoveL 958 to (-91.53, -237.15, -8.35) mm, rotated rx -180 ry 0 rz 0 deg; joints [5.952, -54.331, 125.908, 6.298, -70.81, -1.715]
  MoveC 959 to (-91.98, -237.16, -8.16) mm, rotated rx -180 ry 0 rz 0 deg; joints [5.95, -54.327, 125.872, 6.297, -70.779, -1.718] to (-92.16, -237.16, -7.72) mm, rotated rx -180 ry 0 rz 0 deg; joints [5.949, -54.349, 125.859, 6.297, -70.743, -1.722]
  Set speed (500.0 mm/s)
  MoveL 960 to (-92.16, -237.16, 6) mm, rotated rx 180 ry 0 rz 0 deg; joints [5.945, -55.241, 125.885, 6.327, -69.883, -1.821]
  MoveL 961 to (-92.16, -54.85, 6) mm, rotated rx -180 ry 0 rz 0 deg; joints [14.12, -54.113, 123.31, 15.143, -68.988, -5.052]
  Set speed (25.4 mm/s)
  MoveL 962 to (-92.16, -54.85, -3.54) mm, rotated rx 180 ry 0 rz 0 deg; joints [14.124, -53.515, 123.294, 15.089, -69.55, -4.89]
  MoveC 963 to (-91.98, -54.85, -3.99) mm, rotated rx 180 ry 0 rz 0 deg; joints [14.126, -53.493, 123.308, 15.088, -69.584, -4.881] to (-91.53, -54.85, -4.17) mm, rotated rx -180 ry 0 rz 0 deg; joints [14.131, -53.498, 123.343, 15.091, -69.614, -4.875]
  Set speed (50.8 mm/s)
  MoveL 964 to (-90.89, -54.85, -4.18) mm, rotated rx 180 ry 0 rz 0 deg; joints [14.138, -53.521, 123.394, 15.096, -69.641, -4.87]
  MoveC 965 to (-90.44, -55.04, -4.17) mm, rotated rx 180 ry 0 rz 0 deg; joints [14.135, -53.539, 123.433, 15.09, -69.661, -4.863] to (-90.26, -55.49, -4.17) mm, rotated rx 180 ry 0 rz 0 deg; joints [14.117, -53.55, 123.456, 15.07, -69.672, -4.853]
  MoveL 966 to (-90.26, -80.89, -4.17) mm, rotated rx -180 ry 0 rz 0 deg; joints [13.003, -53.761, 123.94, 13.862, -69.84, -4.388]
  MoveL 967 to (-141.06, -80.89, -4.18) mm, rotated rx -180 ry 0 rz 0 deg; joints [12.506, -51.863, 119.867, 13.531, -67.685, -4.756]
  MoveL 968 to (-141.06, -30.09, -4.17) mm, rotated rx -180 ry 0 rz 0 deg; joints [14.645, -51.423, 118.873, 15.893, -67.356, -5.756]
  MoveL 969 to (-90.26, -30.09, -4.17) mm, rotated rx -180 ry 0 rz 0 deg; joints [15.22, -53.32, 122.932, 16.272, -69.492, -5.33]
  MoveL 970 to (-90.26, -55.49, -4.17) mm, rotated rx 180 ry 0 rz 0 deg; joints [14.117, -53.55, 123.456, 15.07, -69.672, -4.853]
  MoveC 971 to (-90.44, -55.94, -4.18) mm, rotated rx -180 ry 0 rz 0 deg; joints [14.096, -53.547, 123.451, 15.047, -69.667, -4.846] to (-90.89, -56.12, -4.17) mm, rotated rx 180 ry 0 rz 0 deg; joints [14.083, -53.532, 123.419, 15.035, -69.649, -4.846]
  MoveL 972 to (-91.53, -56.12, -4.17) mm, rotated rx -180 ry 0 rz 0 deg; joints [14.076, -53.509, 123.369, 15.03, -69.623, -4.851]
  MoveC 973 to (-91.98, -56.12, -3.99) mm, rotated rx -180 ry 0 rz 0 deg; joints [14.071, -53.504, 123.333, 15.028, -69.593, -4.858] to (-92.16, -56.12, -3.54) mm, rotated rx -180 ry 0 rz 0 deg; joints [14.068, -53.526, 123.32, 15.029, -69.559, -4.867]
  Set speed (500.0 mm/s)
  MoveL 974 to (-92.16, -56.12, 5) mm, rotated rx 180 ry 0 rz 0 deg; joints [14.065, -54.061, 123.334, 15.077, -69.055, -5.01]
  MoveL 975 to (-92.16, -54.85, 5) mm, rotated rx 180 ry 0 rz 0 deg; joints [14.121, -54.05, 123.309, 15.137, -69.047, -5.035]
  Set speed (25.4 mm/s)
  MoveL 976 to (-92.16, -54.85, 1.83) mm, rotated rx 180 ry 0 rz 0 deg; joints [14.122, -53.851, 123.304, 15.119, -69.234, -4.981]
  MoveL 977 to (-92.16, -54.85, -7.71) mm, rotated rx -180 ry 0 rz 0 deg; joints [14.125, -53.252, 123.285, 15.067, -69.795, -4.821]
  MoveC 978 to (-91.98, -54.85, -8.16) mm, rotated rx 180 ry 0 rz 0 deg; joints [14.128, -53.23, 123.299, 15.066, -69.829, -4.812] to (-91.53, -54.85, -8.35) mm, rotated rx -180 ry 0 rz 0 deg; joints [14.133, -53.235, 123.334, 15.068, -69.859, -4.805]
  Set speed (50.8 mm/s)
  MoveL 979 to (-90.89, -54.85, -8.35) mm, rotated rx -180 ry 0 rz 0 deg; joints [14.14, -53.258, 123.384, 15.073, -69.886, -4.8]
  MoveC 980 to (-90.44, -55.04, -8.35) mm, rotated rx 180 ry 0 rz 0 deg; joints [14.136, -53.276, 123.423, 15.067, -69.906, -4.793] to (-90.26, -55.49, -8.35) mm, rotated rx -180 ry 0 rz 0 deg; joints [14.119, -53.287, 123.447, 15.048, -69.917, -4.783]
  MoveL 981 to (-90.26, -80.89, -8.35) mm, rotated rx 180 ry 0 rz 0 deg; joints [13.005, -53.496, 123.93, 13.841, -70.089, -4.324]
  MoveL 982 to (-141.06, -80.89, -8.35) mm, rotated rx -180 ry 0 rz 0 deg; joints [12.507, -51.612, 119.858, 13.509, -67.921, -4.695]
  MoveL 983 to (-141.06, -30.09, -8.35) mm, rotated rx 180 ry 0 rz 0 deg; joints [14.647, -51.174, 118.864, 15.868, -67.586, -5.686]
  MoveL 984 to (-90.26, -30.09, -8.35) mm, rotated rx -180 ry 0 rz 0 deg; joints [15.222, -53.058, 122.923, 16.247, -69.734, -5.255]
  MoveL 985 to (-90.26, -55.49, -8.35) mm, rotated rx -180 ry 0 rz 0 deg; joints [14.119, -53.287, 123.447, 15.048, -69.917, -4.783]
  MoveC 986 to (-90.44, -55.94, -8.35) mm, rotated rx -180 ry 0 rz 0 deg; joints [14.097, -53.284, 123.441, 15.025, -69.912, -4.777] to (-90.89, -56.12, -8.35) mm, rotated rx -180 ry 0 rz 0 deg; joints [14.084, -53.269, 123.409, 15.013, -69.895, -4.777]
  MoveL 987 to (-91.53, -56.12, -8.35) mm, rotated rx -180 ry 0 rz 0 deg; joints [14.077, -53.246, 123.359, 15.008, -69.868, -4.782]
  MoveC 988 to (-91.98, -56.12, -8.16) mm, rotated rx -180 ry 0 rz 0 deg; joints [14.072, -53.241, 123.324, 15.006, -69.838, -4.788] to (-92.16, -56.12, -7.72) mm, rotated rx 180 ry 0 rz 0 deg; joints [14.07, -53.263, 123.31, 15.007, -69.804, -4.797]
  Set speed (500.0 mm/s)
  MoveL 989 to (-92.16, -56.12, 6) mm, rotated rx -180 ry 0 rz 0 deg; joints [14.065, -54.124, 123.335, 15.083, -68.996, -5.027]
  MoveL 990 to (-219.16, -54.85, 6) mm, rotated rx -180 ry 0 rz 0 deg; joints [12.851, -49.157, 112.914, 14.372, -63.598, -6.03]
  Set speed (25.4 mm/s)
  MoveL 991 to (-219.16, -54.85, -3.54) mm, rotated rx 180 ry 0 rz 0 deg; joints [12.854, -48.629, 112.9, 14.313, -64.095, -5.889]
  MoveC 992 to (-218.98, -54.85, -3.99) mm, rotated rx 180 ry 0 rz 0 deg; joints [12.856, -48.612, 112.914, 14.311, -64.127, -5.881] to (-218.53, -54.85, -4.17) mm, rotated rx 180 ry 0 rz 0 deg; joints [12.86, -48.619, 112.952, 14.312, -64.156, -5.875]
  Set speed (50.8 mm/s)
  MoveL 993 to (-217.89, -54.85, -4.18) mm, rotated rx 180 ry 0 rz 0 deg; joints [12.866, -48.645, 113.006, 14.315, -64.185, -5.87]
  MoveC 994 to (-217.44, -55.04, -4.18) mm, rotated rx -180 ry 0 rz 0 deg; joints [12.863, -48.665, 113.048, 14.309, -64.206, -5.862] to (-217.26, -55.49, -4.18) mm, rotated rx 180 ry 0 rz 0 deg; joints [12.847, -48.676, 113.072, 14.289, -64.217, -5.851]
  MoveL 995 to (-217.26, -80.89, -4.18) mm, rotated rx -180 ry 0 rz 0 deg; joints [11.827, -48.887, 113.543, 13.134, -64.364, -5.31]
  MoveL 996 to (-268.06, -80.89, -4.18) mm, rotated rx -180 ry 0 rz 0 deg; joints [11.413, -46.809, 109.162, 12.934, -62.079, -5.69]
  MoveL 997 to (-268.06, -30.09, -4.18) mm, rotated rx -180 ry 0 rz 0 deg; joints [13.378, -46.365, 108.183, 15.217, -61.785, -6.849]
  MoveL 998 to (-217.26, -30.09, -4.17) mm, rotated rx -180 ry 0 rz 0 deg; joints [13.859, -48.446, 112.562, 15.442, -64.058, -6.403]
  MoveL 999 to (-217.26, -55.49, -4.18) mm, rotated rx 180 ry 0 rz 0 deg; joints [12.847, -48.676, 113.072, 14.289, -64.217, -5.851]
  MoveC 1000 to (-217.44, -55.94, -4.18) mm, rotated rx -180 ry 0 rz 0 deg; joints [12.827, -48.672, 113.065, 14.268, -64.211, -5.843] to (-217.89, -56.12, -4.17) mm, rotated rx 180 ry 0 rz 0 deg; joints [12.815, -48.656, 113.031, 14.257, -64.192, -5.843]
  MoveL 1001 to (-218.53, -56.12, -4.17) mm, rotated rx -180 ry 0 rz 0 deg; joints [12.81, -48.63, 112.977, 14.254, -64.164, -5.848]
  MoveC 1002 to (-218.98, -56.12, -3.99) mm, rotated rx 180 ry 0 rz 0 deg; joints [12.806, -48.623, 112.939, 14.253, -64.135, -5.854] to (-219.16, -56.12, -3.54) mm, rotated rx -180 ry 0 rz 0 deg; joints [12.804, -48.64, 112.924, 14.255, -64.103, -5.862]
  Set speed (500.0 mm/s)
  MoveL 1003 to (-219.16, -56.12, 5) mm, rotated rx 180 ry 0 rz 0 deg; joints [12.801, -49.113, 112.938, 14.308, -63.657, -5.987]
  MoveL 1004 to (-219.16, -54.85, 5) mm, rotated rx 180 ry 0 rz 0 deg; joints [12.852, -49.102, 112.913, 14.366, -63.65, -6.015]
  Set speed (25.4 mm/s)
  MoveL 1005 to (-219.16, -54.85, 1.82) mm, rotated rx -180 ry 0 rz 0 deg; joints [12.853, -48.927, 112.909, 14.346, -63.816, -5.968]
  MoveL 1006 to (-219.16, -54.85, -7.72) mm, rotated rx -180 ry 0 rz 0 deg; joints [12.856, -48.397, 112.891, 14.288, -64.312, -5.829]
  MoveC 1007 to (-218.98, -54.85, -8.16) mm, rotated rx 180 ry 0 rz 0 deg; joints [12.858, -48.379, 112.905, 14.286, -64.344, -5.821] to (-218.53, -54.85, -8.35) mm, rotated rx -180 ry 0 rz 0 deg; joints [12.862, -48.387, 112.943, 14.287, -64.373, -5.814]
  Set speed (50.8 mm/s)
  MoveL 1008 to (-217.89, -54.85, -8.35) mm, rotated rx -180 ry 0 rz 0 deg; joints [12.868, -48.412, 112.997, 14.29, -64.401, -5.809]
  MoveC 1009 to (-217.44, -55.04, -8.35) mm, rotated rx -180 ry 0 rz 0 deg; joints [12.864, -48.432, 113.039, 14.284, -64.422, -5.802] to (-217.26, -55.49, -8.35) mm, rotated rx 180 ry 0 rz 0 deg; joints [12.848, -48.443, 113.063, 14.264, -64.433, -5.791]
  MoveL 1010 to (-217.26, -80.89, -8.35) mm, rotated rx -180 ry 0 rz 0 deg; joints [11.828, -48.653, 113.534, 13.111, -64.584, -5.254]
  MoveL 1011 to (-268.06, -80.89, -8.35) mm, rotated rx -180 ry 0 rz 0 deg; joints [11.414, -46.586, 109.153, 12.911, -62.288, -5.637]
  MoveL 1012 to (-268.06, -30.09, -8.35) mm, rotated rx 180 ry 0 rz 0 deg; joints [13.38, -46.144, 108.174, 15.189, -61.99, -6.787]
  MoveL 1013 to (-217.26, -30.09, -8.35) mm, rotated rx -180 ry 0 rz 0 deg; joints [13.86, -48.214, 112.553, 15.414, -64.273, -6.338]
  MoveL 1014 to (-217.26, -55.49, -8.35) mm, rotated rx 180 ry 0 rz 0 deg; joints [12.848, -48.443, 113.063, 14.264, -64.433, -5.791]
  MoveC 1015 to (-217.44, -55.94, -8.35) mm, rotated rx -180 ry 0 rz 0 deg; joints [12.828, -48.44, 113.056, 14.243, -64.428, -5.783] to (-217.89, -56.12, -8.35) mm, rotated rx -180 ry 0 rz 0 deg; joints [12.817, -48.423, 113.022, 14.233, -64.409, -5.782]
  MoveL 1016 to (-218.53, -56.12, -8.35) mm, rotated rx -180 ry 0 rz 0 deg; joints [12.811, -48.398, 112.968, 14.229, -64.381, -5.787]
  MoveC 1017 to (-218.98, -56.12, -8.16) mm, rotated rx -180 ry 0 rz 0 deg; joints [12.807, -48.39, 112.93, 14.228, -64.351, -5.794] to (-219.16, -56.12, -7.72) mm, rotated rx -180 ry 0 rz 0 deg; joints [12.805, -48.408, 112.915, 14.23, -64.32, -5.802]
  Set speed (500.0 mm/s)
  MoveL 1018 to (-219.16, -56.12, 6) mm, rotated rx -180 ry 0 rz 0 deg; joints [12.801, -49.169, 112.939, 14.314, -63.605, -6.002]
  MoveL 1019 to (-346.16, -54.85, 6) mm, rotated rx 180 ry 0 rz 0 deg; joints [11.789, -43.727, 101.648, 13.963, -57.813, -7.091]
  Set speed (25.4 mm/s)
  MoveL 1020 to (-346.16, -54.85, -3.54) mm, rotated rx -180 ry 0 rz 0 deg; joints [11.792, -43.254, 101.634, 13.897, -58.258, -6.963]
  MoveC 1021 to (-345.98, -54.85, -3.99) mm, rotated rx -180 ry 0 rz 0 deg; joints [11.793, -43.24, 101.65, 13.895, -58.288, -6.955] to (-345.53, -54.85, -4.17) mm, rotated rx -180 ry 0 rz 0 deg; joints [11.797, -43.251, 101.692, 13.894, -58.318, -6.948]
  Set speed (50.8 mm/s)
  MoveL 1022 to (-344.89, -54.85, -4.18) mm, rotated rx -180 ry 0 rz 0 deg; joints [11.801, -43.279, 101.751, 13.895, -58.349, -6.943]
  MoveC 1023 to (-344.44, -55.04, -4.18) mm, rotated rx -180 ry 0 rz 0 deg; joints [11.798, -43.3, 101.796, 13.888, -58.371, -6.934] to (-344.26, -55.49, -4.17) mm, rotated rx -180 ry 0 rz 0 deg; joints [11.783, -43.313, 101.822, 13.868, -58.383, -6.921]
  MoveL 1024 to (-344.26, -80.89, -4.17) mm, rotated rx 180 ry 0 rz 0 deg; joints [10.843, -43.529, 102.293, 12.737, -58.518, -6.293]
  MoveL 1025 to (-395.06, -80.89, -4.18) mm, rotated rx 180 ry 0 rz 0 deg; joints [10.493, -41.217, 97.479, 12.678, -56.036, -6.73]
  MoveL 1026 to (-395.06, -30.09, -4.17) mm, rotated rx 180 ry 0 rz 0 deg; joints [12.31, -40.757, 96.486, 14.939, -55.761, -8.075]
  MoveL 1027 to (-344.26, -30.09, -4.17) mm, rotated rx -180 ry 0 rz 0 deg; joints [12.717, -43.077, 101.31, 14.998, -58.237, -7.559]
  MoveL 1028 to (-344.26, -55.49, -4.17) mm, rotated rx -180 ry 0 rz 0 deg; joints [11.783, -43.313, 101.822, 13.868, -58.383, -6.921]
  MoveC 1029 to (-344.44, -55.94, -4.17) mm, rotated rx -180 ry 0 rz 0 deg; joints [11.765, -43.308, 101.813, 13.848, -58.376, -6.912] to (-344.89, -56.12, -4.18) mm, rotated rx -180 ry 0 rz 0 deg; joints [11.755, -43.29, 101.775, 13.839, -58.356, -6.911]
  MoveL 1030 to (-345.53, -56.12, -4.18) mm, rotated rx -180 ry 0 rz 0 deg; joints [11.75, -43.262, 101.716, 13.838, -58.325, -6.917]
  MoveC 1031 to (-345.98, -56.12, -3.99) mm, rotated rx -180 ry 0 rz 0 deg; joints [11.746, -43.251, 101.675, 13.838, -58.295, -6.923] to (-346.16, -56.12, -3.54) mm, rotated rx -180 ry 0 rz 0 deg; joints [11.745, -43.265, 101.658, 13.841, -58.265, -6.931]
  Set speed (500.0 mm/s)
  MoveL 1032 to (-346.16, -56.12, 5) mm, rotated rx -180 ry 0 rz 0 deg; joints [11.742, -43.689, 101.672, 13.899, -57.867, -7.045]
  MoveL 1033 to (-346.16, -54.85, 5) mm, rotated rx -180 ry 0 rz 0 deg; joints [11.789, -43.677, 101.647, 13.956, -57.86, -7.077]
  Set speed (25.4 mm/s)
  MoveL 1034 to (-346.16, -54.85, 1.82) mm, rotated rx 180 ry 0 rz 0 deg; joints [11.79, -43.52, 101.643, 13.934, -58.008, -7.035]
  MoveL 1035 to (-346.16, -54.85, -7.72) mm, rotated rx 180 ry 0 rz 0 deg; joints [11.793, -43.046, 101.625, 13.869, -58.452, -6.907]
  MoveC 1036 to (-345.98, -54.85, -8.16) mm, rotated rx 180 ry 0 rz 0 deg; joints [11.794, -43.032, 101.641, 13.867, -58.482, -6.899] to (-345.53, -54.85, -8.35) mm, rotated rx -180 ry 0 rz 0 deg; joints [11.798, -43.042, 101.683, 13.866, -58.512, -6.893]
  Set speed (50.8 mm/s)
  MoveL 1037 to (-344.89, -54.85, -8.35) mm, rotated rx 180 ry 0 rz 0 deg; joints [11.803, -43.07, 101.742, 13.867, -58.542, -6.887]
  MoveC 1038 to (-344.44, -55.04, -8.35) mm, rotated rx -180 ry 0 rz 0 deg; joints [11.799, -43.092, 101.787, 13.86, -58.565, -6.878] to (-344.26, -55.49, -8.35) mm, rotated rx -180 ry 0 rz 0 deg; joints [11.784, -43.104, 101.813, 13.84, -58.577, -6.866]
  MoveL 1039 to (-344.26, -80.89, -8.35) mm, rotated rx -180 ry 0 rz 0 deg; joints [10.844, -43.319, 102.284, 12.711, -58.714, -6.242]
  MoveL 1040 to (-395.06, -80.89, -8.35) mm, rotated rx -180 ry 0 rz 0 deg; joints [10.494, -41.016, 97.47, 12.651, -56.224, -6.68]
  MoveL 1041 to (-395.06, -30.09, -8.35) mm, rotated rx -180 ry 0 rz 0 deg; joints [12.311, -40.558, 96.477, 14.907, -55.945, -8.017]
  MoveL 1042 to (-344.26, -30.09, -8.35) mm, rotated rx -180 ry 0 rz 0 deg; joints [12.718, -42.87, 101.301, 14.968, -58.429, -7.5]
  MoveL 1043 to (-344.26, -55.49, -8.35) mm, rotated rx -180 ry 0 rz 0 deg; joints [11.784, -43.104, 101.813, 13.84, -58.577, -6.866]
  MoveC 1044 to (-344.44, -55.94, -8.35) mm, rotated rx -180 ry 0 rz 0 deg; joints [11.766, -43.1, 101.804, 13.82, -58.57, -6.856] to (-344.89, -56.12, -8.35) mm, rotated rx -180 ry 0 rz 0 deg; joints [11.756, -43.082, 101.766, 13.811, -58.55, -6.856]
  MoveL 1045 to (-345.53, -56.12, -8.35) mm, rotated rx 180 ry 0 rz 0 deg; joints [11.751, -43.053, 101.707, 13.81, -58.519, -6.861]
  MoveC 1046 to (-345.98, -56.12, -8.16) mm, rotated rx -180 ry 0 rz 0 deg; joints [11.748, -43.043, 101.666, 13.81, -58.489, -6.868] to (-346.16, -56.12, -7.72) mm, rotated rx -180 ry 0 rz 0 deg; joints [11.746, -43.057, 101.65, 13.813, -58.459, -6.876]
  Set speed (500.0 mm/s)
  MoveL 1047 to (-346.16, -56.12, 15) mm, rotated rx 180 ry 0 rz 0 deg; joints [11.739, -44.181, 101.68, 13.97, -57.396, -7.182]
  Print: /'2D Contour1'
  Set speed (500.0 mm/s)
  MoveL 1048 to (-12.15, 15.92, 15) mm, rotated rx -180 ry 0 rz 0 deg; joints [18.266, -56.922, 127.919, 19.338, -71.123, -5.918]
  MoveL 1049 to (-12.15, 15.92, 6) mm, rotated rx -180 ry 0 rz 0 deg; joints [18.27, -56.325, 127.911, 19.277, -71.68, -5.714]
  Set speed (25.4 mm/s)
  MoveL 1050 to (-12.15, 15.92, -4.36) mm, rotated rx 180 ry 0 rz 0 deg; joints [18.275, -55.632, 127.893, 19.209, -72.318, -5.482]
  MoveC 1051 to (-12.34, 15.92, -4.81) mm, rotated rx -180 ry 0 rz 0 deg; joints [18.272, -55.596, 127.878, 19.204, -72.338, -5.473] to (-12.79, 15.92, -5) mm, rotated rx -180 ry 0 rz 0 deg; joints [18.266, -55.568, 127.844, 19.198, -72.331, -5.474]
  Set speed (50.8 mm/s)
  MoveL 1052 to (-13.42, 15.92, -5) mm, rotated rx 180 ry 0 rz 0 deg; joints [18.256, -55.546, 127.796, 19.191, -72.306, -5.48]
  MoveC 1053 to (-13.87, 16.1, -5) mm, rotated rx 180 ry 0 rz 0 deg; joints [18.258, -55.528, 127.757, 19.195, -72.286, -5.487] to (-14.06, 16.55, -5) mm, rotated rx 180 ry 0 rz 0 deg; joints [18.275, -55.517, 127.732, 19.214, -72.275, -5.498]
  MoveL 1054 to (-14.06, 168.95, -5) mm, rotated rx -180 ry 0 rz 0 deg; joints [24.788, -53.532, 123.224, 26.354, -70.775, -8.591]
  MoveL 1055 to (-39.46, 168.95, -5) mm, rotated rx -180 ry 0 rz 0 deg; joints [24.319, -52.645, 121.329, 26.021, -69.796, -8.905]
  MoveC 1056 to (-52.16, 156.25, -5) mm, rotated rx -180 ry 0 rz 0 deg; joints [23.581, -52.386, 120.796, 25.288, -69.432, -8.772] to (-64.86, 168.95, -5) mm, rotated rx -180 ry 0 rz 0 deg; joints [23.866, -51.742, 119.405, 25.711, -68.804, -9.219]
  MoveL 1057 to (-90.26, 168.95, -5) mm, rotated rx -180 ry 0 rz 0 deg; joints [23.428, -50.821, 117.452, 25.424, -67.799, -9.534]
  MoveL 1058 to (-166.46, 168.95, -5) mm, rotated rx 180 ry 0 rz 0 deg; joints [22.202, -47.952, 111.397, 24.7, -64.694, -10.496]
  MoveC 1059 to (-179.16, 156.25, -5) mm, rotated rx 180 ry 0 rz 0 deg; joints [21.535, -47.648, 110.774, 24.037, -64.279, -10.339] to (-191.86, 168.95, -5) mm, rotated rx -180 ry 0 rz 0 deg; joints [21.82, -46.957, 109.308, 24.504, -63.627, -10.826]
  MoveL 1060 to (-293.46, 168.95, -5) mm, rotated rx 180 ry 0 rz 0 deg; joints [20.41, -42.758, 100.543, 23.952, -59.174, -12.228]
  MoveC 1061 to (-306.16, 156.25, -5) mm, rotated rx -180 ry 0 rz 0 deg; joints [19.803, -42.402, 99.816, 23.35, -58.704, -12.054] to (-318.86, 168.95, -5) mm, rotated rx 180 ry 0 rz 0 deg; joints [20.084, -41.647, 98.235, 23.876, -58.009, -12.608]
  MoveL 1062 to (-395.06, 168.95, -5) mm, rotated rx -180 ry 0 rz 0 deg; joints [19.164, -38.136, 90.969, 23.817, -54.359, -13.85]
  MoveL 1063 to (-420.46, 168.95, -5) mm, rotated rx -180 ry 0 rz 0 deg; joints [18.875, -36.899, 88.416, 23.86, -53.084, -14.308]
  MoveC 1064 to (-433.16, 156.25, -5) mm, rotated rx 180 ry 0 rz 0 deg; joints [18.319, -36.473, 87.551, 23.318, -52.542, -14.129] to (-445.86, 168.95, -5) mm, rotated rx -180 ry 0 rz 0 deg; joints [18.595, -35.622, 85.786, 23.939, -51.775, -14.795]
  MoveL 1065 to (-471.26, 168.95, -5) mm, rotated rx 180 ry 0 rz 0 deg; joints [18.322, -34.303, 83.072, 24.059, -50.429, -15.316]
  MoveL 1066 to (-471.26, 16.55, -5) mm, rotated rx -180 ry 0 rz 0 deg; joints [13.323, -36.492, 87.702, 17.096, -51.584, -10.341]
  MoveL 1067 to (-14.06, 16.55, -5) mm, rotated rx -180 ry 0 rz 0 deg; joints [18.275, -55.517, 127.732, 19.214, -72.275, -5.498]
  MoveC 1068 to (-13.61, 16.36, -5) mm, rotated rx -180 ry 0 rz 0 deg; joints [18.274, -55.534, 127.771, 19.21, -72.294, -5.49] to (-13.42, 15.92, -5) mm, rotated rx 180 ry 0 rz 0 deg; joints [18.256, -55.546, 127.796, 19.191, -72.306, -5.48]
  MoveL 1069 to (-13.42, 15.28, -5) mm, rotated rx -180 ry 0 rz 0 deg; joints [18.228, -55.552, 127.812, 19.16, -72.311, -5.468]
  MoveC 1070 to (-13.42, 14.83, -4.81) mm, rotated rx -180 ry 0 rz 0 deg; joints [18.208, -55.57, 127.823, 19.14, -72.304, -5.464] to (-13.42, 14.65, -4.37) mm, rotated rx -180 ry 0 rz 0 deg; joints [18.199, -55.602, 127.829, 19.134, -72.278, -5.471]
  Set speed (500.0 mm/s)
  MoveL 1071 to (-13.42, 14.65, 5) mm, rotated rx -180 ry 0 rz 0 deg; joints [18.195, -56.227, 127.845, 19.195, -71.703, -5.679]
  MoveL 1072 to (-12.15, 15.92, 5) mm, rotated rx 180 ry 0 rz 0 deg; joints [18.271, -56.258, 127.91, 19.27, -71.742, -5.691]
  Set speed (25.4 mm/s)
  MoveL 1073 to (-12.15, 15.92, 1) mm, rotated rx -180 ry 0 rz 0 deg; joints [18.273, -55.991, 127.904, 19.244, -71.988, -5.601]
  MoveL 1074 to (-12.15, 15.92, -7.71) mm, rotated rx 180 ry 0 rz 0 deg; joints [18.276, -55.408, 127.885, 19.188, -72.522, -5.407]
  MoveC 1075 to (-12.34, 15.92, -8.16) mm, rotated rx -180 ry 0 rz 0 deg; joints [18.274, -55.371, 127.87, 19.183, -72.542, -5.399] to (-12.79, 15.92, -8.35) mm, rotated rx -180 ry 0 rz 0 deg; joints [18.267, -55.343, 127.836, 19.177, -72.536, -5.399]
  Set speed (50.8 mm/s)
  MoveL 1076 to (-13.42, 15.92, -8.35) mm, rotated rx -180 ry 0 rz 0 deg; joints [18.258, -55.321, 127.788, 19.17, -72.51, -5.406]
  MoveC 1077 to (-13.87, 16.1, -8.35) mm, rotated rx 180 ry 0 rz 0 deg; joints [18.26, -55.304, 127.749, 19.174, -72.49, -5.413] to (-14.06, 16.55, -8.35) mm, rotated rx -180 ry 0 rz 0 deg; joints [18.277, -55.292, 127.724, 19.193, -72.479, -5.423]
  MoveL 1078 to (-14.06, 168.95, -8.35) mm, rotated rx 180 ry 0 rz 0 deg; joints [24.79, -53.321, 123.217, 26.324, -70.957, -8.496]
  MoveL 1079 to (-39.46, 168.95, -8.35) mm, rotated rx -180 ry 0 rz 0 deg; joints [24.32, -52.439, 121.322, 25.99, -69.974, -8.813]
  MoveC 1080 to (-52.16, 156.25, -8.35) mm, rotated rx -180 ry 0 rz 0 deg; joints [23.583, -52.182, 120.788, 25.258, -69.61, -8.683] to (-64.86, 168.95, -8.35) mm, rotated rx 180 ry 0 rz 0 deg; joints [23.867, -51.541, 119.398, 25.68, -68.979, -9.129]
  MoveL 1081 to (-90.26, 168.95, -8.35) mm, rotated rx -180 ry 0 rz 0 deg; joints [23.43, -50.625, 117.444, 25.393, -67.969, -9.447]
  MoveL 1082 to (-166.46, 168.95, -8.35) mm, rotated rx -180 ry 0 rz 0 deg; joints [22.203, -47.769, 111.389, 24.667, -64.854, -10.415]
  MoveC 1083 to (-179.16, 156.25, -8.35) mm, rotated rx 180 ry 0 rz 0 deg; joints [21.537, -47.466, 110.767, 24.004, -64.439, -10.261] to (-191.86, 168.95, -8.35) mm, rotated rx -180 ry 0 rz 0 deg; joints [21.821, -46.778, 109.301, 24.47, -63.784, -10.747]
  MoveL 1084 to (-293.46, 168.95, -8.35) mm, rotated rx 180 ry 0 rz 0 deg; joints [20.411, -42.593, 100.536, 23.915, -59.319, -12.154]
  MoveC 1085 to (-306.16, 156.25, -8.35) mm, rotated rx -180 ry 0 rz 0 deg; joints [19.804, -42.237, 99.809, 23.314, -58.849, -11.982] to (-318.86, 168.95, -8.35) mm, rotated rx -180 ry 0 rz 0 deg; joints [20.085, -41.485, 98.228, 23.838, -58.151, -12.534]
  MoveL 1086 to (-395.06, 168.95, -8.35) mm, rotated rx -180 ry 0 rz 0 deg; joints [19.165, -37.983, 90.962, 23.776, -54.493, -13.778]
  MoveL 1087 to (-420.46, 168.95, -8.35) mm, rotated rx -180 ry 0 rz 0 deg; joints [18.876, -36.748, 88.409, 23.818, -53.216, -14.237]
  MoveC 1088 to (-433.16, 156.25, -8.35) mm, rotated rx 180 ry 0 rz 0 deg; joints [18.32, -36.324, 87.543, 23.276, -52.673, -14.059] to (-445.86, 168.95, -8.35) mm, rotated rx -180 ry 0 rz 0 deg; joints [18.596, -35.474, 85.779, 23.896, -51.904, -14.724]
  MoveL 1089 to (-471.26, 168.95, -8.35) mm, rotated rx -180 ry 0 rz 0 deg; joints [18.323, -34.157, 83.065, 24.014, -50.556, -15.244]
  MoveL 1090 to (-471.26, 16.55, -8.35) mm, rotated rx -180 ry 0 rz 0 deg; joints [13.324, -36.342, 87.695, 17.064, -51.72, -10.289]
  MoveL 1091 to (-14.06, 16.55, -8.35) mm, rotated rx -180 ry 0 rz 0 deg; joints [18.277, -55.292, 127.724, 19.193, -72.479, -5.423]
  MoveC 1092 to (-13.61, 16.36, -8.35) mm, rotated rx 180 ry 0 rz 0 deg; joints [18.275, -55.31, 127.763, 19.189, -72.499, -5.416] to (-13.42, 15.92, -8.35) mm, rotated rx -180 ry 0 rz 0 deg; joints [18.258, -55.321, 127.788, 19.17, -72.51, -5.406]
  MoveL 1093 to (-13.42, 15.28, -8.35) mm, rotated rx -180 ry 0 rz 0 deg; joints [18.23, -55.328, 127.804, 19.139, -72.516, -5.394]
  MoveC 1094 to (-13.42, 14.83, -8.16) mm, rotated rx -180 ry 0 rz 0 deg; joints [18.209, -55.345, 127.815, 19.119, -72.508, -5.39] to (-13.42, 14.65, -7.72) mm, rotated rx -180 ry 0 rz 0 deg; joints [18.201, -55.377, 127.821, 19.113, -72.483, -5.396]
  Set speed (500.0 mm/s)
  MoveL 1095 to (-13.42, 14.65, 6) mm, rotated rx 180 ry 0 rz 0 deg; joints [18.195, -56.293, 127.847, 19.201, -71.641, -5.702]
  MoveL 1096 to (18.41, 14.65, 6) mm, rotated rx 180 ry 0 rz 0 deg; joints [18.674, -57.413, 130.234, 19.567, -72.885, -5.405]
  Set speed (25.4 mm/s)
  MoveL 1097 to (18.41, 14.65, -4.36) mm, rotated rx 180 ry 0 rz 0 deg; joints [18.679, -56.697, 130.216, 19.501, -73.543, -5.163]
  MoveC 1098 to (18.41, 14.83, -4.81) mm, rotated rx -180 ry 0 rz 0 deg; joints [18.687, -56.664, 130.21, 19.508, -73.57, -5.156] to (18.41, 15.28, -5) mm, rotated rx 180 ry 0 rz 0 deg; joints [18.708, -56.646, 130.198, 19.529, -73.578, -5.159]
  Set speed (50.8 mm/s)
  MoveL 1099 to (18.41, 15.92, -5) mm, rotated rx 180 ry 0 rz 0 deg; joints [18.737, -56.639, 130.182, 19.559, -73.572, -5.171]
  MoveC 1100 to (18.6, 16.36, -5) mm, rotated rx 180 ry 0 rz 0 deg; joints [18.76, -56.641, 130.185, 19.584, -73.575, -5.177] to (19.05, 16.55, -5) mm, rotated rx -180 ry 0 rz 0 deg; joints [18.776, -56.654, 130.213, 19.598, -73.591, -5.176]
  MoveL 1101 to (39.46, 16.55, -5) mm, rotated rx -180 ry 0 rz 0 deg; joints [19.098, -57.342, 131.724, 19.852, -74.396, -4.974]
  MoveL 1102 to (471.26, 16.55, -5) mm, rotated rx -180 ry 0 rz 30 deg; joints [37.425, -66.202, 151.706, 67.551, -87.389, -4.354]
  MoveL 1103 to (471.26, 168.95, -5) mm, rotated rx -180 ry 0 rz 0 deg; joints [38.476, -67.383, 154.732, 38.527, -87.056, -1.378]
  MoveL 1104 to (445.86, 168.95, -5) mm, rotated rx -180 ry 0 rz 0 deg; joints [37.447, -66.819, 153.298, 37.528, -86.337, -1.872]
  MoveC 1105 to (433.16, 156.25, -5) mm, rotated rx -180 ry 0 rz 0 deg; joints [36.291, -66.724, 153.115, 36.373, -86.223, -1.867] to (420.46, 168.95, -5) mm, rotated rx -180 ry 0 rz 0 deg; joints [36.464, -66.234, 151.838, 36.58, -85.598, -2.346]
  MoveL 1106 to (395.06, 168.95, -5) mm, rotated rx 180 ry 0 rz 0 deg; joints [35.525, -65.628, 150.354, 35.682, -84.841, -2.802]
  MoveL 1107 to (318.86, 168.95, -5) mm, rotated rx -180 ry 0 rz 0 deg; joints [32.945, -63.698, 145.757, 33.26, -82.475, -4.074]
  MoveC 1108 to (306.16, 156.25, -5) mm, rotated rx 180 ry 0 rz 0 deg; joints [31.926, -63.559, 145.469, 32.245, -82.273, -4.034] to (293.46, 168.95, -5) mm, rotated rx -180 ry 0 rz 0 deg; joints [32.158, -63.019, 144.178, 32.535, -81.657, -4.47]
  MoveL 1109 to (191.86, 168.95, -5) mm, rotated rx -180 ry 0 rz 0 deg; joints [29.32, -60.138, 137.637, 30.003, -78.256, -5.942]
  MoveC 1110 to (179.16, 156.25, -5) mm, rotated rx 180 ry 0 rz 0 deg; joints [28.418, -59.955, 137.257, 29.106, -77.988, -5.866] to (166.46, 168.95, -5) mm, rotated rx -180 ry 0 rz 0 deg; joints [28.681, -59.378, 135.944, 29.453, -77.376, -6.288]
  MoveL 1111 to (90.26, 168.95, -5) mm, rotated rx 180 ry 0 rz 0 deg; joints [26.908, -57.005, 130.727, 27.98, -74.663, -7.285]
  MoveL 1112 to (64.86, 168.95, -5) mm, rotated rx -180 ry 0 rz 0 deg; joints [26.362, -56.184, 128.94, 27.544, -73.735, -7.608]
  MoveC 1113 to (61.14, 159.97, -5) mm, rotated rx 180 ry 0 rz 0 deg; joints [25.9, -56.199, 128.988, 27.063, -73.702, -7.465] to (52.16, 156.25, -5) mm, rotated rx -180 ry 0 rz 0 deg; joints [25.556, -55.959, 128.476, 26.745, -73.412, -7.499]
  MoveL 1114 to (52.16, 156.25, -5) mm, rotated rx -180 ry 0 rz 0 deg; joints [25.556, -55.959, 128.476, 26.745, -73.412, -7.499]
  MoveC 1115 to (43.18, 159.97, -5) mm, rotated rx -180 ry 0 rz 0 deg; joints [25.532, -55.606, 127.705, 26.776, -73.035, -7.688] to (39.46, 168.95, -5) mm, rotated rx -180 ry 0 rz 0 deg; joints [25.835, -55.347, 127.128, 27.135, -72.795, -7.927]
  MoveL 1116 to (14.06, 168.95, -5) mm, rotated rx 180 ry 0 rz 0 deg; joints [25.328, -54.494, 125.29, 26.75, -71.843, -8.243]
  MoveL 1117 to (14.06, 16.55, -5) mm, rotated rx -180 ry 0 rz 0 deg; joints [18.699, -56.484, 129.842, 19.538, -73.394, -5.225]
  MoveL 1118 to (19.05, 16.55, -5) mm, rotated rx -180 ry 0 rz 0 deg; joints [18.776, -56.654, 130.213, 19.598, -73.591, -5.176]
  MoveC 1119 to (19.49, 16.36, -5) mm, rotated rx 180 ry 0 rz 0 deg; joints [18.774, -56.671, 130.251, 19.595, -73.611, -5.168] to (19.68, 15.92, -5) mm, rotated rx -180 ry 0 rz 0 deg; joints [18.757, -56.682, 130.277, 19.575, -73.622, -5.158]
  MoveL 1120 to (19.68, 15.28, -5) mm, rotated rx 180 ry 0 rz 0 deg; joints [18.728, -56.689, 130.293, 19.544, -73.628, -5.147]
  MoveC 1121 to (19.68, 14.83, -4.81) mm, rotated rx 180 ry 0 rz 0 deg; joints [18.707, -56.707, 130.304, 19.523, -73.62, -5.143] to (19.68, 14.65, -4.37) mm, rotated rx -180 ry 0 rz 0 deg; joints [18.698, -56.74, 130.31, 19.517, -73.594, -5.15]
  Set speed (500.0 mm/s)
  MoveL 1122 to (19.68, 14.65, 5) mm, rotated rx -180 ry 0 rz 0 deg; joints [18.694, -57.389, 130.327, 19.576, -72.998, -5.37]
  MoveL 1123 to (18.41, 14.65, 5) mm, rotated rx -180 ry 0 rz 0 deg; joints [18.674, -57.344, 130.232, 19.56, -72.949, -5.382]
  Set speed (25.4 mm/s)
  MoveL 1124 to (18.41, 14.65, 1) mm, rotated rx -180 ry 0 rz 0 deg; joints [18.676, -57.068, 130.226, 19.535, -73.203, -5.288]
  MoveL 1125 to (18.41, 14.65, -7.72) mm, rotated rx 180 ry 0 rz 0 deg; joints [18.68, -56.464, 130.208, 19.481, -73.755, -5.085]
  MoveC 1126 to (18.41, 14.83, -8.16) mm, rotated rx -180 ry 0 rz 0 deg; joints [18.689, -56.431, 130.202, 19.487, -73.782, -5.078] to (18.41, 15.28, -8.35) mm, rotated rx 180 ry 0 rz 0 deg; joints [18.709, -56.414, 130.19, 19.508, -73.789, -5.082]
  Set speed (50.8 mm/s)
  MoveL 1127 to (18.41, 15.92, -8.35) mm, rotated rx -180 ry 0 rz 0 deg; joints [18.738, -56.407, 130.174, 19.539, -73.783, -5.093]
  MoveC 1128 to (18.6, 16.36, -8.35) mm, rotated rx -180 ry 0 rz 0 deg; joints [18.762, -56.408, 130.176, 19.563, -73.787, -5.099] to (19.05, 16.55, -8.35) mm, rotated rx -180 ry 0 rz 0 deg; joints [18.777, -56.421, 130.205, 19.578, -73.803, -5.098]
  MoveL 1129 to (39.46, 16.55, -8.35) mm, rotated rx -180 ry 0 rz 0 deg; joints [19.099, -57.104, 131.716, 19.832, -74.612, -4.893]
  MoveL 1130 to (471.26, 16.55, -8.35) mm, rotated rx -180 ry 0 rz 30 deg; joints [37.428, -65.85, 151.696, 67.54, -87.519, -4.039]
  MoveL 1131 to (471.26, 168.95, -8.35) mm, rotated rx -180 ry 0 rz 0 deg; joints [38.479, -67.002, 154.721, 38.519, -87.345, -1.148]
  MoveL 1132 to (445.86, 168.95, -8.35) mm, rotated rx -180 ry 0 rz 0 deg; joints [37.45, -66.452, 153.287, 37.517, -86.618, -1.655]
  MoveC 1133 to (433.16, 156.25, -8.35) mm, rotated rx -180 ry 0 rz 0 deg; joints [36.294, -66.359, 153.104, 36.363, -86.507, -1.657] to (420.46, 168.95, -8.35) mm, rotated rx 180 ry 0 rz 0 deg; joints [36.467, -65.881, 151.827, 36.568, -85.873, -2.141]
  MoveL 1134 to (395.06, 168.95, -8.35) mm, rotated rx -180 ry 0 rz 0 deg; joints [35.527, -65.288, 150.343, 35.668, -85.109, -2.609]
  MoveL 1135 to (318.86, 168.95, -8.35) mm, rotated rx -180 ry 0 rz 0 deg; joints [32.947, -63.391, 145.747, 33.241, -82.723, -3.91]
  MoveC 1136 to (306.16, 156.25, -8.35) mm, rotated rx -180 ry 0 rz 0 deg; joints [31.928, -63.254, 145.459, 32.227, -82.523, -3.875] to (293.46, 168.95, -8.35) mm, rotated rx 180 ry 0 rz 0 deg; joints [32.16, -62.722, 144.169, 32.515, -81.899, -4.314]
  MoveL 1137 to (191.86, 168.95, -8.35) mm, rotated rx -180 ry 0 rz 0 deg; joints [29.323, -59.876, 137.628, 29.979, -78.476, -5.813]
  MoveC 1138 to (179.16, 156.25, -8.35) mm, rotated rx -180 ry 0 rz 0 deg; joints [28.42, -59.695, 137.248, 29.082, -78.208, -5.742] to (166.46, 168.95, -8.35) mm, rotated rx -180 ry 0 rz 0 deg; joints [28.683, -59.123, 135.936, 29.428, -77.59, -6.164]
  MoveL 1139 to (90.26, 168.95, -8.35) mm, rotated rx 180 ry 0 rz 0 deg; joints [26.91, -56.771, 130.719, 27.953, -74.863, -7.176]
  MoveL 1140 to (64.86, 168.95, -8.35) mm, rotated rx 180 ry 0 rz 0 deg; joints [26.364, -55.956, 128.932, 27.516, -73.93, -7.502]
  MoveC 1141 to (61.14, 159.97, -8.35) mm, rotated rx 180 ry 0 rz 0 deg; joints [25.902, -55.97, 128.98, 27.036, -73.898, -7.361] to (52.16, 156.25, -8.35) mm, rotated rx -180 ry 0 rz 0 deg; joints [25.558, -55.733, 128.468, 26.717, -73.607, -7.397]
  MoveL 1142 to (52.16, 156.25, -8.35) mm, rotated rx 180 ry 0 rz 0 deg; joints [25.558, -55.733, 128.468, 26.717, -73.607, -7.397]
  MoveC 1143 to (43.18, 159.97, -8.35) mm, rotated rx -180 ry 0 rz 0 deg; joints [25.534, -55.382, 127.697, 26.748, -73.228, -7.587] to (39.46, 168.95, -8.35) mm, rotated rx -180 ry 0 rz 0 deg; joints [25.837, -55.124, 127.12, 27.106, -72.986, -7.825]
  MoveL 1144 to (14.06, 168.95, -8.35) mm, rotated rx -180 ry 0 rz 0 deg; joints [25.33, -54.277, 125.282, 26.721, -72.03, -8.145]
  MoveL 1145 to (14.06, 16.55, -8.35) mm, rotated rx 180 ry 0 rz 0 deg; joints [18.7, -56.253, 129.834, 19.518, -73.604, -5.147]
  MoveL 1146 to (19.05, 16.55, -8.35) mm, rotated rx -180 ry 0 rz 0 deg; joints [18.777, -56.421, 130.205, 19.578, -73.803, -5.098]
  MoveC 1147 to (19.49, 16.36, -8.35) mm, rotated rx 180 ry 0 rz 0 deg; joints [18.776, -56.438, 130.243, 19.574, -73.822, -5.09] to (19.68, 15.92, -8.35) mm, rotated rx -180 ry 0 rz 0 deg; joints [18.758, -56.45, 130.268, 19.554, -73.834, -5.08]
  MoveL 1148 to (19.68, 15.28, -8.35) mm, rotated rx -180 ry 0 rz 0 deg; joints [18.729, -56.456, 130.284, 19.524, -73.84, -5.069]
  MoveC 1149 to (19.68, 14.83, -8.16) mm, rotated rx 180 ry 0 rz 0 deg; joints [18.708, -56.474, 130.296, 19.503, -73.832, -5.066] to (19.68, 14.65, -7.72) mm, rotated rx -180 ry 0 rz 0 deg; joints [18.7, -56.507, 130.302, 19.496, -73.806, -5.073]
  Set speed (500.0 mm/s)
  MoveL 1150 to (19.68, 14.65, 6) mm, rotated rx -180 ry 0 rz 0 deg; joints [18.694, -57.458, 130.328, 19.582, -72.934, -5.393]
  MoveL 1151 to (12.15, -16.75, 6) mm, rotated rx 180 ry 0 rz 0 deg; joints [17.138, -57.528, 130.524, 17.95, -72.906, -4.899]
  Set speed (25.4 mm/s)
  MoveL 1152 to (12.15, -16.75, -4.37) mm, rotated rx -180 ry 0 rz 0 deg; joints [17.143, -56.808, 130.505, 17.89, -73.573, -4.675]
  MoveC 1153 to (12.34, -16.75, -4.81) mm, rotated rx -180 ry 0 rz 0 deg; joints [17.146, -56.784, 130.518, 17.89, -73.609, -4.664] to (12.79, -16.75, -5) mm, rotated rx 180 ry 0 rz 0 deg; joints [17.152, -56.786, 130.551, 17.894, -73.639, -4.656]
  Set speed (50.8 mm/s)
  MoveL 1154 to (13.42, -16.75, -5) mm, rotated rx -180 ry 0 rz 0 deg; joints [17.161, -56.808, 130.599, 17.901, -73.665, -4.65]
  MoveC 1155 to (13.87, -16.94, -5) mm, rotated rx -180 ry 0 rz 0 deg; joints [17.159, -56.825, 130.637, 17.897, -73.684, -4.643] to (14.06, -17.39, -5) mm, rotated rx -180 ry 0 rz 0 deg; joints [17.141, -56.836, 130.661, 17.877, -73.696, -4.634]
  MoveL 1156 to (14.06, -169.79, -5) mm, rotated rx -180 ry 0 rz 0 deg; joints [9.847, -57.999, 133.431, 10.203, -74.783, -2.282]
  MoveL 1157 to (471.26, -169.79, -5) mm, rotated rx -180 ry 0 rz -60 deg; joints [-6.05, -67.111, 155.762, -66.063, -89.254, 2.122]
  MoveL 1158 to (471.26, -17.39, -5) mm, rotated rx -180 ry 0 rz -60 deg; joints [4.313, -67.251, 155.931, -55.702, -89.057, 1.98]
  MoveL 1159 to (445.86, -17.39, -5) mm, rotated rx -180 ry 0 rz -60 deg; joints [4.187, -66.591, 154.123, -55.849, -88.415, 2.932]
